KUKA KRL program: MyProgram_317().src

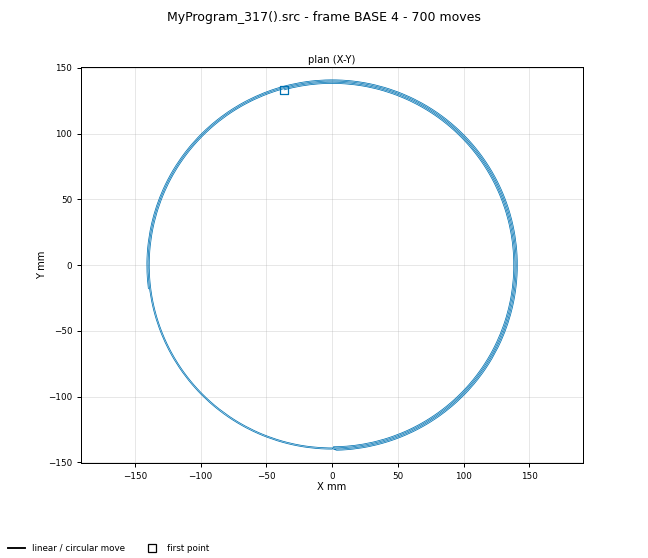
[picture p0: tool path of MyProgram_317().src in frame BASE 4, 700 of 700 moves have a stored position in this frame; points joined in program order, loops and branches not executed]
&ACCESS RVP
&REL 1
&PARAM TEMPLATE = C:\KRC\Roboter\Template\vorgabe
&PARAM EDITMASK = *
DEF MyProgram_317()
; ---- Setting reference (Base) ----
$BASE = BASE_DATA[4]

; --------------------------
; ---- Setting tool (TCP) ----
$TOOL = TOOL_DATA[3]
; --------------------------

$VEL.CP = VEL_APROX_PRINT
Startdeposition()
$VEL.CP = VEL_PRINT
LIN {X -36.4177,Y 133.3267,Z 184,A 105.8748,B 3.6775,C 0.0605,E1 3.6399,E2 347.4823} C_DIS
LIN {X -33.6227,Y 134.0568,Z 184,A 104.6666,B 3.6776,C 0.0598,E1 3.6432,E2 348.691} C_DIS
LIN {X -29.9714,Y 134.9221,Z 184,A 103.1035,B 3.6776,C 0.059,E1 3.6474,E2 350.2543} C_DIS
LIN {X -26.7547,Y 135.5966,Z 184,A 101.734,B 3.6776,C 0.0584,E1 3.6512,E2 351.6239} C_DIS
LIN {X -23.5921,Y 136.1822,Z 184,A 100.3951,B 3.6776,C 0.0579,E1 3.6549,E2 352.9627} C_DIS
LIN {X -20.3485,Y 136.7048,Z 184,A 99.029,B 3.6776,C 0.0575,E1 3.6586,E2 354.3286} C_DIS
LIN {X -17.2099,Y 137.135,Z 184,A 97.7126,B 3.6776,C 0.0572,E1 3.6623,E2 355.6447} C_DIS
LIN {X -14.2664,Y 137.4713,Z 184,A 96.4709,B 3.6776,C 0.057,E1 3.6657,E2 356.8874} C_DIS
LIN {X -10.8915,Y 137.7809,Z 184,A 95.0782,B 3.6776,C 0.0567,E1 3.6696,E2 358.278} C_DIS
LIN {X -7.7622,Y 137.9925,Z 184,A 93.7791,B 3.6776,C 0.0566,E1 3.6732,E2 359.5763} C_DIS
LIN {X -3.6918,Y 138.1595,Z 184,A 92.0273,B 3.6776,C 0.0571,E1 3.6781,E2 361.3349} C_DIS
LIN {X 0,Y 138.2109,Z 184,A 90.5659,B 3.6776,C 0.0566,E1 3.6822,E2 362.7873} C_DIS
LIN {X 3.0237,Y 138.1776,Z 184,A 89.3114,B 3.6776,C 0.0568,E1 3.6857,E2 364.0415} C_DIS
LIN {X 6.1171,Y 138.0752,Z 184,A 88.0293,B 3.6776,C 0.0571,E1 3.6893,E2 365.3229} C_DIS
LIN {X 10.3123,Y 137.8236,Z 184,A 86.2404,B 3.6776,C 0.0579,E1 3.6943,E2 367.1167} C_DIS
LIN {X 13.9962,Y 137.5004,Z 184,A 84.7627,B 3.6776,C 0.058,E1 3.6984,E2 368.5872} C_DIS
LIN {X 17.1189,Y 137.1464,Z 184,A 83.4643,B 3.6776,C 0.0585,E1 3.702,E2 369.8846} C_DIS
LIN {X 20.3485,Y 136.7048,Z 184,A 82.1206,B 3.6776,C 0.0591,E1 3.7057,E2 371.227} C_DIS
LIN {X 23.0597,Y 136.2716,Z 184,A 80.9465,B 3.6776,C 0.0601,E1 3.7089,E2 372.405} C_DIS
LIN {X 26.7088,Y 135.6054,Z 184,A 79.462,B 3.6776,C 0.0606,E1 3.713,E2 373.8826} C_DIS
LIN {X 29.9253,Y 134.932,Z 184,A 78.1102,B 3.6776,C 0.0614,E1 3.7167,E2 375.2327} C_DIS
LIN {X 32.8099,Y 134.2582,Z 184,A 76.899,B 3.6776,C 0.0622,E1 3.72,E2 376.4414} C_DIS
LIN {X 35.9709,Y 133.4458,Z 184,A 75.5188,B 3.6776,C 0.0635,E1 3.7237,E2 377.8247} C_DIS
LIN {X 39.6415,Y 132.404,Z 184,A 73.9879,B 3.6776,C 0.0644,E1 3.7278,E2 379.3491} C_DIS
LIN {X 42.8155,Y 131.4116,Z 184,A 72.6248,B 3.6776,C 0.0656,E1 3.7314,E2 380.7099} C_DIS
LIN {X 45.6313,Y 130.4587,Z 184,A 71.4074,B 3.6775,C 0.0667,E1 3.7346,E2 381.9252} C_DIS
LIN {X 49.2779,Y 129.1276,Z 184,A 69.8203,B 3.6775,C 0.0682,E1 3.7388,E2 383.5094} C_DIS
LIN {X 52.4222,Y 127.8831,Z 184,A 68.4385,B 3.6775,C 0.0696,E1 3.7424,E2 384.8886} C_DIS
LIN {X 55.1838,Y 126.7138,Z 184,A 67.1766,B 3.6774,C 0.0713,E1 3.7456,E2 386.1525} C_DIS
LIN {X 58.7493,Y 125.1027,Z 184,A 65.6176,B 3.6774,C 0.0727,E1 3.7495,E2 387.7036} C_DIS
LIN {X 61.8796,Y 123.5843,Z 184,A 64.203,B 3.6774,C 0.0744,E1 3.7531,E2 389.1147} C_DIS
LIN {X 64.8421,Y 122.0551,Z 184,A 62.835,B 3.6773,C 0.0761,E1 3.7565,E2 390.4809} C_DIS
LIN {X 68.469,Y 120.0586,Z 184,A 61.0927,B 3.6773,C 0.0789,E1 3.7607,E2 392.2263} C_DIS
LIN {X 71.8734,Y 118.0527,Z 184,A 59.5538,B 3.6773,C 0.0804,E1 3.7644,E2 393.753} C_DIS
LIN {X 74.8883,Y 116.1637,Z 184,A 58.1092,B 3.6772,C 0.0824,E1 3.7678,E2 395.1939} C_DIS
LIN {X 77.8197,Y 114.2206,Z 184,A 56.6827,B 3.6772,C 0.0845,E1 3.7711,E2 396.6165} C_DIS
LIN {X 80.7488,Y 112.169,Z 184,A 55.2381,B 3.6771,C 0.0867,E1 3.7744,E2 398.0564} C_DIS
LIN {X 83.9195,Y 109.8161,Z 184,A 53.5602,B 3.677,C 0.0899,E1 3.7781,E2 399.7395} C_DIS
LIN {X 87.1141,Y 107.3005,Z 184,A 51.9899,B 3.677,C 0.0918,E1 3.7815,E2 401.2957} C_DIS
LIN {X 90.0725,Y 104.8286,Z 184,A 50.3385,B 3.6769,C 0.0954,E1 3.7851,E2 402.9538} C_DIS
LIN {X 93.2043,Y 102.055,Z 184,A 48.7445,B 3.6769,C 0.0973,E1 3.7883,E2 404.5307} C_DIS
LIN {X 95.7956,Y 99.6265,Z 184,A 47.3082,B 3.6767,C 0.0999,E1 3.7912,E2 405.9628} C_DIS
LIN {X 98.6354,Y 96.8148,Z 184,A 45.6237,B 3.6767,C 0.1035,E1 3.7946,E2 407.6509} C_DIS
LIN {X 101.4499,Y 93.8625,Z 184,A 44.0571,B 3.6766,C 0.1058,E1 3.7975,E2 409.2025} C_DIS
LIN {X 104.0652,Y 90.9534,Z 184,A 42.3981,B 3.6765,C 0.1097,E1 3.8006,E2 410.8664} C_DIS
LIN {X 106.7196,Y 87.8247,Z 184,A 40.8296,B 3.6764,C 0.112,E1 3.8034,E2 412.4188} C_DIS
LIN {X 108.9505,Y 85.0413,Z 184,A 39.4004,B 3.6763,C 0.1148,E1 3.8059,E2 413.8423} C_DIS
LIN {X 111.2875,Y 81.9584,Z 184,A 37.7496,B 3.6762,C 0.119,E1 3.8086,E2 415.4993} C_DIS
LIN {X 113.7044,Y 78.572,Z 184,A 36.1718,B 3.6761,C 0.1215,E1 3.8111,E2 417.0593} C_DIS
LIN {X 115.668,Y 75.6515,Z 184,A 34.6865,B 3.676,C 0.1252,E1 3.8134,E2 418.5484} C_DIS
LIN {X 118.0397,Y 71.895,Z 184,A 32.9814,B 3.6759,C 0.1282,E1 3.8159,E2 420.237} C_DIS
LIN {X 119.8206,Y 68.8859,Z 184,A 31.5781,B 3.6757,C 0.1313,E1 3.8179,E2 421.635} C_DIS
LIN {X 121.5433,Y 65.7989,Z 184,A 30.0427,B 3.6756,C 0.1357,E1 3.82,E2 423.1798} C_DIS
LIN {X 123.5623,Y 61.9243,Z 184,A 28.4136,B 3.6755,C 0.1383,E1 3.822,E2 424.7867} C_DIS
LIN {X 125.0605,Y 58.8392,Z 184,A 27.0414,B 3.6754,C 0.1414,E1 3.8237,E2 426.1533} C_DIS
LIN {X 126.3707,Y 55.9663,Z 184,A 25.7977,B 3.6753,C 0.1441,E1 3.8251,E2 427.3892} C_DIS
LIN {X 127.7,Y 52.8622,Z 184,A 24.3996,B 3.6751,C 0.1477,E1 3.8266,E2 428.7878} C_DIS
LIN {X 129.1276,Y 49.2779,Z 184,A 22.8878,B 3.675,C 0.151,E1 3.8281,E2 430.2893} C_DIS
LIN {X 130.2884,Y 46.1206,Z 184,A 21.5479,B 3.6749,C 0.1541,E1 3.8294,E2 431.6229} C_DIS
LIN {X 131.2362,Y 43.3441,Z 184,A 20.3532,B 3.6747,C 0.1571,E1 3.8304,E2 432.8155} C_DIS
LIN {X 132.404,Y 39.6415,Z 184,A 18.8234,B 3.6746,C 0.1606,E1 3.8317,E2 434.3361} C_DIS
LIN {X 133.3267,Y 36.4177,Z 184,A 17.4858,B 3.6744,C 0.1638,E1 3.8327,E2 435.6678} C_DIS
LIN {X 134.0348,Y 33.7096,Z 184,A 16.324,B 3.6743,C 0.167,E1 3.8335,E2 436.8304} C_DIS
LIN {X 134.9221,Y 29.9714,Z 184,A 14.837,B 3.6742,C 0.1702,E1 3.8344,E2 438.3049} C_DIS
LIN {X 135.5966,Y 26.7547,Z 184,A 13.5266,B 3.674,C 0.1734,E1 3.8352,E2 439.6095} C_DIS
LIN {X 136.1822,Y 23.5921,Z 184,A 12.2445,B 3.6739,C 0.1765,E1 3.8358,E2 440.8858} C_DIS
LIN {X 136.7048,Y 20.3485,Z 184,A 10.9352,B 3.6737,C 0.1797,E1 3.8363,E2 442.1892} C_DIS
LIN {X 137.0724,Y 17.6872,Z 184,A 9.8194,B 3.6735,C 0.1829,E1 3.8368,E2 443.3059} C_DIS
LIN {X 137.4956,Y 14.0415,Z 184,A 8.4072,B 3.6734,C 0.1859,E1 3.8372,E2 444.7052} C_DIS
LIN {X 137.7809,Y 10.8915,Z 184,A 7.1428,B 3.6732,C 0.1891,E1 3.8375,E2 445.9645} C_DIS
LIN {X 137.9925,Y 7.7622,Z 184,A 5.9051,B 3.6731,C 0.192,E1 3.8377,E2 447.195} C_DIS
LIN {X 138.1604,Y 3.6595,Z 184,A 4.2009,B 3.6728,C 0.1969,E1 3.8379,E2 448.9004} C_DIS
LIN {X 138.2105,Y 0,Z 184,A 2.8172,B 3.6727,C 0.1996,E1 3.8379,E2 450.2682} C_DIS
LIN {X 138.1769,Y -3.0677,Z 184,A 1.5727,B 3.6725,C 0.2029,E1 3.8379,E2 451.51} C_DIS
LIN {X 138.0752,Y -6.1171,Z 184,A 0.3524,B 3.6723,C 0.206,E1 3.8377,E2 452.7255} C_DIS
LIN {X 137.8237,Y -10.3111,Z 184,A -1.3754,B 3.6721,C 0.2107,E1 3.8374,E2 454.4526} C_DIS
LIN {X 137.5004,Y -13.9962,Z 184,A -2.8057,B 3.6719,C 0.2139,E1 3.837,E2 455.8708} C_DIS
LIN {X 137.1464,Y -17.1189,Z 184,A -4.063,B 3.6717,C 0.217,E1 3.8366,E2 457.1232} C_DIS
LIN {X 136.7048,Y -20.3485,Z 184,A -5.3655,B 3.6715,C 0.2203,E1 3.8361,E2 458.4205} C_DIS
LIN {X 136.2752,Y -23.0383,Z 184,A -6.4989,B 3.6713,C 0.2235,E1 3.8356,E2 459.5551} C_DIS
LIN {X 135.6054,Y -26.7088,Z 184,A -7.9465,B 3.6711,C 0.2267,E1 3.8348,E2 460.9911} C_DIS
LIN {X 134.932,Y -29.9253,Z 184,A -9.2568,B 3.6709,C 0.2299,E1 3.8341,E2 462.2958} C_DIS
LIN {X 134.1769,Y -33.1472,Z 184,A -10.5844,B 3.6707,C 0.2332,E1 3.8332,E2 463.6187} C_DIS
LIN {X 133.4627,Y -35.9077,Z 184,A -11.7334,B 3.6705,C 0.236,E1 3.8324,E2 464.7642} C_DIS
LIN {X 132.4869,Y -39.3583,Z 184,A -13.1732,B 3.6703,C 0.2396,E1 3.8313,E2 466.1992} C_DIS
LIN {X 131.4116,Y -42.8155,Z 184,A -14.6088,B 3.6701,C 0.2429,E1 3.8301,E2 467.6275} C_DIS
LIN {X 130.3049,Y -46.0747,Z 184,A -15.9862,B 3.6699,C 0.2462,E1 3.8288,E2 468.9996} C_DIS
LIN {X 129.1276,Y -49.2779,Z 184,A -17.3523,B 3.6696,C 0.2494,E1 3.8275,E2 470.3606} C_DIS
LIN {X 127.9871,Y -52.1642,Z 184,A -18.6113,B 3.6694,C 0.2525,E1 3.8262,E2 471.617} C_DIS
LIN {X 126.5358,Y -55.5957,Z 184,A -20.0872,B 3.6692,C 0.2558,E1 3.8246,E2 473.0852} C_DIS
LIN {X 125.276,Y -58.3747,Z 184,A -21.3124,B 3.669,C 0.2586,E1 3.8231,E2 474.3062} C_DIS
LIN {X 123.5843,Y -61.8796,Z 184,A -22.8693,B 3.6687,C 0.2621,E1 3.8212,E2 475.8571} C_DIS
LIN {X 121.9809,Y -64.9833,Z 184,A -24.2702,B 3.6685,C 0.2653,E1 3.8194,E2 477.2531} C_DIS
LIN {X 120.2686,Y -68.1009,Z 184,A -25.6961,B 3.6683,C 0.2685,E1 3.8175,E2 478.6738} C_DIS
LIN {X 118.5194,Y -71.1011,Z 184,A -27.1792,B 3.668,C 0.2725,E1 3.8154,E2 480.1638} C_DIS
LIN {X 116.1637,Y -74.8883,Z 184,A -28.8795,B 3.6678,C 0.2754,E1 3.8128,E2 481.8462} C_DIS
LIN {X 114.2206,Y -77.8197,Z 184,A -30.2911,B 3.6676,C 0.2784,E1 3.8107,E2 483.253} C_DIS
LIN {X 112.169,Y -80.7488,Z 184,A -31.7282,B 3.6673,C 0.2814,E1 3.8083,E2 484.6853} C_DIS
LIN {X 109.8667,Y -83.8533,Z 184,A -33.3715,B 3.667,C 0.2855,E1 3.8056,E2 486.3352} C_DIS
LIN {X 107.3005,Y -87.1141,Z 184,A -35.0216,B 3.6668,C 0.2887,E1 3.8027,E2 487.9776} C_DIS
LIN {X 104.4481,Y -90.5143,Z 184,A -36.7357,B 3.6665,C 0.2914,E1 3.7996,E2 489.6767} C_DIS
LIN {X 102.055,Y -93.2043,Z 184,A -38.2644,B 3.6663,C 0.295,E1 3.7968,E2 491.2114} C_DIS
LIN {X 98.9867,Y -96.4567,Z 184,A -40.0606,B 3.666,C 0.2983,E1 3.7933,E2 493.0015} C_DIS
LIN {X 95.8325,Y -99.591,Z 184,A -41.7813,B 3.6658,C 0.3008,E1 3.7899,E2 494.7077} C_DIS
LIN {X 93.2043,Y -102.055,Z 184,A -43.2299,B 3.6656,C 0.3033,E1 3.7869,E2 496.1515} C_DIS
LIN {X 90.1903,Y -104.7271,Z 184,A -44.9204,B 3.6653,C 0.3068,E1 3.7834,E2 497.846} C_DIS
LIN {X 87.1339,Y -107.2843,Z 184,A -46.4677,B 3.6651,C 0.3088,E1 3.7801,E2 499.3809} C_DIS
LIN {X 84.317,Y -109.5121,Z 184,A -47.9844,B 3.6649,C 0.3118,E1 3.7767,E2 500.9024} C_DIS
LIN {X 80.7694,Y -112.1541,Z 184,A -49.6964,B 3.6647,C 0.3138,E1 3.7729,E2 502.5998} C_DIS
LIN {X 77.8407,Y -114.2063,Z 184,A -51.1541,B 3.6645,C 0.3161,E1 3.7695,E2 504.0554} C_DIS
LIN {X 74.8883,Y -116.1637,Z 184,A -52.5889,B 3.6643,C 0.3182,E1 3.7662,E2 505.4868} C_DIS
LIN {X 71.895,Y -118.0397,Z 184,A -54.0208,B 3.6641,C 0.3202,E1 3.7628,E2 506.9156} C_DIS
LIN {X 68.8859,Y -119.8206,Z 184,A -55.4417,B 3.664,C 0.3221,E1 3.7594,E2 508.3337} C_DIS
LIN {X 65.6732,Y -121.6108,Z 184,A -57.0582,B 3.6637,C 0.3253,E1 3.7554,E2 509.9635} C_DIS
LIN {X 61.9243,Y -123.5623,Z 184,A -58.6521,B 3.6637,C 0.3262,E1 3.7515,E2 511.5378} C_DIS
LIN {X 58.8392,Y -125.0605,Z 184,A -60.0471,B 3.6635,C 0.3278,E1 3.748,E2 512.9302} C_DIS
LIN {X 55.641,Y -126.5161,Z 184,A -61.4766,B 3.6633,C 0.3294,E1 3.7443,E2 514.3572} C_DIS
LIN {X 52.4678,Y -127.8647,Z 184,A -62.881,B 3.6632,C 0.3309,E1 3.7407,E2 515.7593} C_DIS
LIN {X 49.2779,Y -129.1276,Z 184,A -64.2795,B 3.6631,C 0.3323,E1 3.7371,E2 517.1556} C_DIS
LIN {X 46.1206,Y -130.2884,Z 184,A -65.6513,B 3.6629,C 0.3336,E1 3.7335,E2 518.5253} C_DIS
LIN {X 43.3085,Y -131.2481,Z 184,A -66.8658,B 3.6629,C 0.3347,E1 3.7303,E2 519.7384} C_DIS
LIN {X 39.6415,Y -132.404,Z 184,A -68.4354,B 3.6627,C 0.336,E1 3.7261,E2 521.3058} C_DIS
LIN {X 36.4177,Y -133.3267,Z 184,A -69.8062,B 3.6627,C 0.3371,E1 3.7224,E2 522.675} C_DIS
LIN {X 33.1934,Y -134.1658,Z 184,A -71.1697,B 3.6625,C 0.3381,E1 3.7187,E2 524.037} C_DIS
LIN {X 30.4533,Y -134.812,Z 184,A -72.3636,B 3.6625,C 0.3392,E1 3.7154,E2 525.2351} C_DIS
LIN {X 26.7547,Y -135.5966,Z 184,A -73.8726,B 3.6624,C 0.3398,E1 3.7113,E2 526.7373} C_DIS
LIN {X 23.5921,Y -136.1822,Z 184,A -75.1907,B 3.6624,C 0.3405,E1 3.7077,E2 528.0542} C_DIS
LIN {X 20.3485,Y -136.7048,Z 184,A -76.541,B 3.6622,C 0.3412,E1 3.704,E2 529.4037} C_DIS
LIN {X 17.2099,Y -137.135,Z 184,A -77.8367,B 3.6622,C 0.3417,E1 3.7004,E2 530.6977} C_DIS
LIN {X 14.5476,Y -137.4411,Z 184,A -78.9933,B 3.6622,C 0.3426,E1 3.6971,E2 531.861} C_DIS
LIN {X 10.8915,Y -137.7809,Z 184,A -80.4558,B 3.6622,C 0.3427,E1 3.6931,E2 533.3165} C_DIS
LIN {X 7.7622,Y -137.9925,Z 184,A -81.7476,B 3.6621,C 0.3431,E1 3.6895,E2 534.6078} C_DIS
LIN {X 4.6115,Y -138.134,Z 184,A -83.048,B 3.6621,C 0.3433,E1 3.6859,E2 535.9079} C_DIS
LIN {X 0.9865,Y -138.204,Z 184,A -84.071,B 3.6624,C 0.3395,E1 3.6832,E2 536.8675} C_DIS
Enddeposition()
LIN {X 0.9865,Y -138.204,Z 184,A -84.071,B 3.6624,C 0.3395,E1 3.6832,E2 536.8675} C_DIS
Startdeposition()
$VEL.CP = VEL_PRINT
LIN {X 1.6267,Y -139.1018,Z 184,A -83.626,B 3.6446,C 0.3393,E1 3.6667,E2 536.434} C_DIS
LIN {X 4.5561,Y -139.0367,Z 184,A -82.3295,B 3.6447,C 0.3382,E1 3.6703,E2 535.1247} C_DIS
LIN {X 8.311,Y -138.8613,Z 184,A -81.0351,B 3.6446,C 0.34,E1 3.6738,E2 533.8639} C_DIS
LIN {X 11.0661,Y -138.6702,Z 184,A -79.683,B 3.6448,C 0.3376,E1 3.6777,E2 532.4822} C_DIS
LIN {X 14.8601,Y -138.3135,Z 184,A -78.2274,B 3.6448,C 0.338,E1 3.6817,E2 531.0411} C_DIS
LIN {X 22.3175,Y -137.3087,Z 184,A -75.1897,B 3.6448,C 0.3369,E1 3.6901,E2 528.0102} C_DIS
LIN {X 27.2301,Y -136.4192,Z 184,A -73.0374,B 3.6451,C 0.3346,E1 3.696,E2 525.8436} C_DIS
LIN {X 31.257,Y -135.5525,Z 184,A -71.0765,B 3.6454,C 0.3308,E1 3.7015,E2 523.8458} C_DIS
LIN {X 34.8949,Y -134.6633,Z 184,A -69.7728,B 3.6454,C 0.3318,E1 3.7049,E2 522.5736} C_DIS
LIN {X 38.7466,Y -133.6046,Z 184,A -68.4032,B 3.6452,C 0.3329,E1 3.7085,E2 521.2402} C_DIS
LIN {X 42.0447,Y -132.6035,Z 184,A -66.8695,B 3.6454,C 0.3305,E1 3.7127,E2 519.6902} C_DIS
LIN {X 45.813,Y -131.3491,Z 184,A -64.552,B 3.6462,C 0.3221,E1 3.719,E2 517.2789} C_DIS
LIN {X 51.2002,Y -129.346,Z 184,A -62.7921,B 3.6459,C 0.3253,E1 3.7234,E2 515.6001} C_DIS
LIN {X 54.8124,Y -127.8558,Z 184,A -61.4097,B 3.6459,C 0.3256,E1 3.7269,E2 514.2473} C_DIS
LIN {X 57.5864,Y -126.6329,Z 184,A -59.9335,B 3.6462,C 0.3218,E1 3.7307,E2 512.7395} C_DIS
LIN {X 60.8952,Y -125.0744,Z 184,A -58.6873,B 3.6462,C 0.3223,E1 3.7338,E2 511.5274} C_DIS
LIN {X 63.9287,Y -123.5522,Z 184,A -57.1271,B 3.6465,C 0.3187,E1 3.7377,E2 509.9442} C_DIS
LIN {X 67.7295,Y -121.5103,Z 184,A -55.4455,B 3.6466,C 0.3171,E1 3.7418,E2 508.2743} C_DIS
LIN {X 71.3493,Y -119.4202,Z 184,A -53.9193,B 3.6466,C 0.3164,E1 3.7454,E2 506.7731} C_DIS
LIN {X 75.2493,Y -117.0022,Z 184,A -51.9472,B 3.647,C 0.3126,E1 3.7501,E2 504.7885} C_DIS
LIN {X 78.5811,Y -114.7908,Z 184,A -50.3195,B 3.6472,C 0.31,E1 3.7539,E2 503.1621} C_DIS
LIN {X 81.9197,Y -112.433,Z 184,A -48.5917,B 3.6475,C 0.3066,E1 3.7578,E2 501.427} C_DIS
LIN {X 86.4283,Y -109.0051,Z 184,A -46.356,B 3.6478,C 0.3033,E1 3.7627,E2 499.2025} C_DIS
LIN {X 89.6043,Y -106.4097,Z 184,A -44.7166,B 3.648,C 0.3007,E1 3.7662,E2 497.5686} C_DIS
LIN {X 92.8185,Y -103.6176,Z 184,A -43.0112,B 3.6483,C 0.2977,E1 3.7698,E2 495.8682} C_DIS
LIN {X 96.4701,Y -100.2276,Z 184,A -41.08,B 3.6485,C 0.2949,E1 3.7737,E2 493.9516} C_DIS
LIN {X 99.1485,Y -97.5783,Z 184,A -39.5527,B 3.6487,C 0.2919,E1 3.7767,E2 492.4263} C_DIS
LIN {X 101.875,Y -94.7279,Z 184,A -37.9879,B 3.6489,C 0.2891,E1 3.7797,E2 490.8682} C_DIS
LIN {X 104.0406,Y -92.3445,Z 184,A -36.5334,B 3.6493,C 0.2848,E1 3.7824,E2 489.3954} C_DIS
LIN {X 107.3985,Y -88.4172,Z 184,A -34.5568,B 3.6495,C 0.2818,E1 3.7859,E2 487.4374} C_DIS
LIN {X 110.2779,Y -84.7985,Z 184,A -32.9995,B 3.6495,C 0.2812,E1 3.7886,E2 485.925} C_DIS
LIN {X 113.183,Y -80.8795,Z 184,A -30.7961,B 3.6501,C 0.2744,E1 3.7922,E2 483.694} C_DIS
LIN {X 115.3285,Y -77.79,Z 184,A -29.2513,B 3.6504,C 0.2707,E1 3.7947,E2 482.1486} C_DIS
LIN {X 117.9246,Y -73.7956,Z 184,A -27.3604,B 3.6506,C 0.2668,E1 3.7975,E2 480.2656} C_DIS
LIN {X 120.0287,Y -70.3209,Z 184,A -25.5164,B 3.6511,C 0.2607,E1 3.8001,E2 478.3973} C_DIS
LIN {X 121.8673,Y -67.0847,Z 184,A -24.3462,B 3.6511,C 0.2609,E1 3.8017,E2 477.2744} C_DIS
LIN {X 123.5248,Y -63.9809,Z 184,A -22.7776,B 3.6514,C 0.2559,E1 3.8037,E2 475.6887} C_DIS
LIN {X 125.4873,Y -60.0356,Z 184,A -21.2126,B 3.6516,C 0.2541,E1 3.8056,E2 474.1553} C_DIS
LIN {X 127.2516,Y -56.2031,Z 184,A -19.4239,B 3.6519,C 0.249,E1 3.8076,E2 472.3585} C_DIS
LIN {X 128.9238,Y -52.25,Z 184,A -17.8419,B 3.6521,C 0.2464,E1 3.8093,E2 470.7998} C_DIS
LIN {X 129.9917,Y -49.5393,Z 184,A -16.3578,B 3.6525,C 0.24,E1 3.8108,E2 469.277} C_DIS
LIN {X 131.2146,Y -46.2011,Z 184,A -15.1434,B 3.6525,C 0.2389,E1 3.8119,E2 468.0946} C_DIS
LIN {X 132.3294,Y -42.9028,Z 184,A -13.9835,B 3.6526,C 0.2381,E1 3.8129,E2 466.9699} C_DIS
LIN {X 133.423,Y -39.3669,Z 184,A -12.4,B 3.6529,C 0.2333,E1 3.8142,E2 465.3774} C_DIS
LIN {X 134.2134,Y -36.5889,Z 184,A -11.3088,B 3.6531,C 0.2312,E1 3.815,E2 464.2983} C_DIS
LIN {X 135.1389,Y -33.0005,Z 184,A -9.7166,B 3.6534,C 0.2262,E1 3.8161,E2 462.6962} C_DIS
LIN {X 136.8507,Y -24.9703,Z 184,A -6.558,B 3.6538,C 0.2194,E1 3.8179,E2 459.5646} C_DIS
LIN {X 137.8292,Y -18.845,Z 184,A -3.9527,B 3.6543,C 0.2117,E1 3.819,E2 456.9508} C_DIS
LIN {X 138.2931,Y -15.0497,Z 184,A -2.6362,B 3.6543,C 0.2102,E1 3.8194,E2 455.667} C_DIS
LIN {X 138.6077,Y -11.8054,Z 184,A -1.2782,B 3.6546,C 0.2062,E1 3.8197,E2 454.3061} C_DIS
LIN {X 138.8743,Y -8.0994,Z 184,A 0.3268,B 3.6549,C 0.2011,E1 3.82,E2 452.6903} C_DIS
LIN {X 139.0413,Y -4.39,Z 184,A 1.5468,B 3.6549,C 0.2003,E1 3.8201,E2 451.5097} C_DIS
LIN {X 139.1063,Y -0.9898,Z 184,A 3.0194,B 3.6552,C 0.1955,E1 3.8201,E2 450.0267} C_DIS
LIN {X 139.0868,Y 2.5321,Z 184,A 4.4683,B 3.6554,C 0.1914,E1 3.8201,E2 448.577} C_DIS
LIN {X 138.9387,Y 6.8925,Z 184,A 6.1187,B 3.6555,C 0.188,E1 3.8199,E2 446.9445} C_DIS
LIN {X 138.7685,Y 9.7424,Z 184,A 7.2364,B 3.6557,C 0.1854,E1 3.8197,E2 445.8337} C_DIS
LIN {X 138.4021,Y 14.031,Z 184,A 9.0908,B 3.656,C 0.1795,E1 3.8193,E2 443.9676} C_DIS
LIN {X 137.8074,Y 19.0003,Z 184,A 11.021,B 3.6562,C 0.1752,E1 3.8186,E2 442.0532} C_DIS
LIN {X 136.6868,Y 25.8495,Z 184,A 13.7424,B 3.6565,C 0.1688,E1 3.8173,E2 439.3479} C_DIS
LIN {X 135.7284,Y 30.4871,Z 184,A 15.6833,B 3.6567,C 0.1635,E1 3.8162,E2 437.4072} C_DIS
LIN {X 134.8596,Y 34.1218,Z 184,A 17.0595,B 3.6568,C 0.1611,E1 3.8153,E2 436.0513} C_DIS
LIN {X 133.9801,Y 37.4261,Z 184,A 18.3557,B 3.6569,C 0.1585,E1 3.8143,E2 434.7687} C_DIS
LIN {X 133.1804,Y 40.1828,Z 184,A 19.6449,B 3.6571,C 0.1541,E1 3.8133,E2 433.4652} C_DIS
LIN {X 132.0698,Y 43.6921,Z 184,A 21.0366,B 3.6572,C 0.1514,E1 3.8121,E2 432.0887} C_DIS
LIN {X 131.1049,Y 46.5121,Z 184,A 22.1652,B 3.6573,C 0.1493,E1 3.8111,E2 430.9723} C_DIS
LIN {X 129.8289,Y 49.9603,Z 184,A 23.702,B 3.6575,C 0.145,E1 3.8095,E2 429.4319} C_DIS
LIN {X 128.518,Y 53.2411,Z 184,A 25.1194,B 3.6576,C 0.1416,E1 3.8081,E2 428.0187} C_DIS
LIN {X 127.0919,Y 56.5602,Z 184,A 26.5206,B 3.6577,C 0.1387,E1 3.8065,E2 426.6279} C_DIS
LIN {X 125.8669,Y 59.241,Z 184,A 27.6711,B 3.6578,C 0.1363,E1 3.8052,E2 425.4851} C_DIS
LIN {X 124.2392,Y 62.5804,Z 184,A 29.2061,B 3.658,C 0.1323,E1 3.8032,E2 423.9489} C_DIS
LIN {X 122.3439,Y 66.2122,Z 184,A 30.8919,B 3.6581,C 0.1281,E1 3.801,E2 422.2627} C_DIS
LIN {X 120.2591,Y 69.9265,Z 184,A 32.5879,B 3.6583,C 0.1244,E1 3.7987,E2 420.5735} C_DIS
LIN {X 117.9197,Y 73.8036,Z 184,A 34.407,B 3.6583,C 0.1204,E1 3.796,E2 418.7597} C_DIS
LIN {X 115.4373,Y 77.6292,Z 184,A 36.2311,B 3.6585,C 0.1165,E1 3.7932,E2 416.9419} C_DIS
LIN {X 112.8595,Y 81.3312,Z 184,A 38.0454,B 3.6586,C 0.1126,E1 3.7903,E2 415.1326} C_DIS
LIN {X 110.3375,Y 84.7206,Z 184,A 40.762,B 3.6591,C 0.0983,E1 3.7855,E2 412.29} C_DIS
LIN {X 105.0956,Y 91.1426,Z 184,A 43.1443,B 3.659,C 0.1018,E1 3.7814,E2 410.0398} C_DIS
LIN {X 101.7038,Y 94.9118,Z 184,A 45.037,B 3.659,C 0.0994,E1 3.7778,E2 408.1715} C_DIS
LIN {X 98.4714,Y 98.2617,Z 184,A 46.909,B 3.6591,C 0.0959,E1 3.7742,E2 406.305} C_DIS
LIN {X 96.221,Y 100.4661,Z 184,A 48.7641,B 3.6593,C 0.0876,E1 3.7703,E2 404.3788} C_DIS
LIN {X 92.093,Y 104.2629,Z 184,A 50.4182,B 3.6593,C 0.0899,E1 3.767,E2 402.8079} C_DIS
LIN {X 88.23,Y 107.5519,Z 184,A 52.4688,B 3.6593,C 0.0864,E1 3.7626,E2 400.762} C_DIS
LIN {X 84.5498,Y 110.4682,Z 184,A 54.3314,B 3.6594,C 0.0836,E1 3.7585,E2 398.9083} C_DIS
LIN {X 81.5522,Y 112.6993,Z 184,A 56.4543,B 3.6596,C 0.0751,E1 3.7536,E2 396.7114} C_DIS
LIN {X 76.8945,Y 115.9272,Z 184,A 58.1486,B 3.6596,C 0.0777,E1 3.7498,E2 395.0982} C_DIS
LIN {X 73.4331,Y 118.1502,Z 184,A 59.7449,B 3.6596,C 0.076,E1 3.7461,E2 393.5143} C_DIS
LIN {X 69.8491,Y 120.3039,Z 184,A 61.4765,B 3.6596,C 0.0733,E1 3.7419,E2 391.7815} C_DIS
LIN {X 65.8036,Y 122.5634,Z 184,A 63.3616,B 3.6596,C 0.0708,E1 3.7373,E2 389.8994} C_DIS
LIN {X 63.0762,Y 123.9868,Z 184,A 65.1665,B 3.6598,C 0.064,E1 3.7326,E2 388.0267} C_DIS
LIN {X 58.1292,Y 126.382,Z 184,A 66.826,B 3.6598,C 0.0668,E1 3.7286,E2 386.4438} C_DIS
LIN {X 53.9781,Y 128.2102,Z 184,A 68.4391,B 3.6598,C 0.067,E1 3.7246,E2 384.8628} C_DIS
LIN {X 51.4322,Y 129.2534,Z 184,A 69.7852,B 3.6598,C 0.0637,E1 3.721,E2 383.4903} C_DIS
LIN {X 47.4222,Y 130.7767,Z 184,A 71.4346,B 3.6598,C 0.0629,E1 3.7167,E2 381.8559} C_DIS
LIN {X 42.7659,Y 132.3731,Z 184,A 73.2656,B 3.6598,C 0.0627,E1 3.7119,E2 380.0499} C_DIS
LIN {X 39.1536,Y 133.4855,Z 184,A 74.85,B 3.6598,C 0.061,E1 3.7077,E2 378.4624} C_DIS
LIN {X 36.3496,Y 134.2772,Z 184,A 76.1941,B 3.6598,C 0.0587,E1 3.704,E2 377.1006} C_DIS
LIN {X 33.0187,Y 135.1345,Z 184,A 77.5771,B 3.6599,C 0.0579,E1 3.7003,E2 375.7222} C_DIS
LIN {X 24.4171,Y 136.9497,Z 184,A 81.1038,B 3.6599,C 0.0564,E1 3.6907,E2 372.2085} C_DIS
LIN {X 18.0552,Y 137.9328,Z 184,A 83.6491,B 3.6599,C 0.056,E1 3.6837,E2 369.6773} C_DIS
LIN {X 15.6018,Y 138.2337,Z 184,A 84.8854,B 3.6599,C 0.0537,E1 3.6802,E2 368.4143} C_DIS
LIN {X 11.7127,Y 138.6155,Z 184,A 86.3851,B 3.6599,C 0.0541,E1 3.676,E2 366.9288} C_DIS
LIN {X 7.8041,Y 138.8925,Z 184,A 87.9522,B 3.6599,C 0.0541,E1 3.6717,E2 365.3682} C_DIS
LIN {X 3.8245,Y 139.057,Z 184,A 89.6538,B 3.6599,C 0.0532,E1 3.6669,E2 363.6596} C_DIS
LIN {X 0.0191,Y 139.1116,Z 184,A 91.3045,B 3.6599,C 0.0523,E1 3.6623,E2 361.9993} C_DIS
LIN {X -3.784,Y 139.0582,Z 184,A 92.7529,B 3.6599,C 0.0532,E1 3.6583,E2 360.5662} C_DIS
LIN {X -10.3027,Y 138.7276,Z 184,A 95.4954,B 3.6599,C 0.053,E1 3.6506,E2 357.8183} C_DIS
LIN {X -15.9841,Y 138.189,Z 184,A 97.9614,B 3.6599,C 0.0526,E1 3.6437,E2 355.3392} C_DIS
LIN {X -20.9141,Y 137.5288,Z 184,A 100.0074,B 3.6599,C 0.0532,E1 3.638,E2 353.2946} C_DIS
LIN {X -25.7351,Y 136.7087,Z 184,A 101.9476,B 3.6599,C 0.0546,E1 3.6327,E2 351.3647} C_DIS
LIN {X -28.779,Y 136.1011,Z 184,A 103.2928,B 3.6599,C 0.0547,E1 3.629,E2 350.0118} C_DIS
LIN {X -33.0872,Y 135.118,Z 184,A 105.1396,B 3.6599,C 0.0556,E1 3.624,E2 348.1628} C_DIS
LIN {X -36.6135,Y 134.2068,Z 184,A 106.5072,B 3.6599,C 0.0575,E1 3.6204,E2 346.8126} C_DIS
LIN {X -40.4202,Y 133.1077,Z 184,A 108.1679,B 3.6599,C 0.0584,E1 3.6159,E2 345.1492} C_DIS
LIN {X -43.7292,Y 132.0575,Z 184,A 109.5897,B 3.6599,C 0.0596,E1 3.6121,E2 343.7292} C_DIS
LIN {X -48.4928,Y 130.3837,Z 184,A 111.881,B 3.6599,C 0.06,E1 3.606,E2 341.413} C_DIS
LIN {X -52.5033,Y 128.8217,Z 184,A 113.5293,B 3.6599,C 0.0625,E1 3.6018,E2 339.7813} C_DIS
LIN {X -56.3097,Y 127.2039,Z 184,A 115.2757,B 3.6599,C 0.064,E1 3.5973,E2 338.0307} C_DIS
LIN {X -59.2446,Y 125.8651,Z 184,A 116.7209,B 3.6598,C 0.0647,E1 3.5936,E2 336.5719} C_DIS
LIN {X -61.9097,Y 124.574,Z 184,A 118.1052,B 3.6598,C 0.0651,E1 3.5901,E2 335.1678} C_DIS
LIN {X -66.5866,Y 122.1397,Z 184,A 120.126,B 3.6598,C 0.0688,E1 3.5852,E2 333.1675} C_DIS
LIN {X -69.3122,Y 120.6147,Z 184,A 121.5354,B 3.6598,C 0.0697,E1 3.5817,E2 331.7437} C_DIS
LIN {X -73.4102,Y 118.1644,Z 184,A 123.4348,B 3.6596,C 0.0729,E1 3.5772,E2 329.854} C_DIS
LIN {X -76.6291,Y 116.1029,Z 184,A 125.0133,B 3.6596,C 0.0752,E1 3.5735,E2 328.2761} C_DIS
LIN {X -80.3195,Y 113.5812,Z 184,A 126.7049,B 3.6596,C 0.079,E1 3.5697,E2 326.6045} C_DIS
LIN {X -86.1401,Y 109.233,Z 184,A 129.7441,B 3.6594,C 0.0836,E1 3.5629,E2 323.5619} C_DIS
LIN {X -88.7601,Y 107.1146,Z 184,A 131.4324,B 3.6594,C 0.0842,E1 3.5592,E2 321.8372} C_DIS
LIN {X -92.3931,Y 103.9976,Z 184,A 133.9759,B 3.6594,C 0.0843,E1 3.5537,E2 319.2231} C_DIS
LIN {X -96.0771,Y 100.6036,Z 184,A 135.5035,B 3.6592,C 0.0914,E1 3.5507,E2 317.7646} C_DIS
LIN {X -98.8636,Y 97.8669,Z 184,A 137.2072,B 3.6592,C 0.094,E1 3.5473,E2 316.0503} C_DIS
LIN {X -102.027,Y 94.5647,Z 184,A 138.9066,B 3.659,C 0.0989,E1 3.5441,E2 314.3754} C_DIS
LIN {X -104.9691,Y 91.2876,Z 184,A 141.0447,B 3.659,C 0.1008,E1 3.5401,E2 312.1981} C_DIS
LIN {X -107.9339,Y 87.7626,Z 184,A 143.0355,B 3.6589,C 0.1043,E1 3.5365,E2 310.197} C_DIS
LIN {X -110.8287,Y 84.0774,Z 184,A 145.0073,B 3.6588,C 0.1084,E1 3.5331,E2 308.2215} C_DIS
LIN {X -113.3153,Y 80.6945,Z 184,A 147.0695,B 3.6588,C 0.1104,E1 3.5297,E2 306.1185} C_DIS
LIN {X -115.5054,Y 77.527,Z 184,A 148.7884,B 3.6586,C 0.1134,E1 3.527,E2 304.384} C_DIS
LIN {X -117.8525,Y 73.9111,Z 184,A 150.269,B 3.6584,C 0.1192,E1 3.5249,E2 302.9423} C_DIS
LIN {X -120.9395,Y 68.7429,Z 184,A 152.769,B 3.6582,C 0.1251,E1 3.5213,E2 300.4417} C_DIS
LIN {X -122.9591,Y 65.0582,Z 184,A 154.4393,B 3.6581,C 0.1297,E1 3.5191,E2 298.7803} C_DIS
LIN {X -124.6141,Y 61.8285,Z 184,A 156.0438,B 3.658,C 0.1329,E1 3.5171,E2 297.1631} C_DIS
LIN {X -126.1958,Y 58.5319,Z 184,A 157.6136,B 3.6578,C 0.1364,E1 3.5152,E2 295.5864} C_DIS
LIN {X -127.4712,Y 55.702,Z 184,A 158.8125,B 3.6577,C 0.1401,E1 3.5139,E2 294.3986} C_DIS
LIN {X -128.8472,Y 52.4401,Z 184,A 160.4985,B 3.6576,C 0.1427,E1 3.512,E2 292.6849} C_DIS
LIN {X -130.1864,Y 49.0195,Z 184,A 161.993,B 3.6574,C 0.1467,E1 3.5105,E2 291.1939} C_DIS
LIN {X -131.4023,Y 45.6597,Z 184,A 163.5458,B 3.6573,C 0.1502,E1 3.5091,E2 289.6319} C_DIS
LIN {X -132.4494,Y 42.5273,Z 184,A 164.9571,B 3.6571,C 0.1536,E1 3.5079,E2 288.2151} C_DIS
LIN {X -133.3363,Y 39.6632,Z 184,A 166.2226,B 3.6571,C 0.1568,E1 3.5068,E2 286.9467} C_DIS
LIN {X -134.3484,Y 36.0826,Z 184,A 167.8458,B 3.6569,C 0.1605,E1 3.5056,E2 285.3131} C_DIS
LIN {X -135.1557,Y 32.9311,Z 184,A 169.0778,B 3.6567,C 0.1647,E1 3.5048,E2 284.096} C_DIS
LIN {X -135.8758,Y 29.823,Z 184,A 170.6517,B 3.6566,C 0.167,E1 3.5038,E2 282.4898} C_DIS
LIN {X -136.6192,Y 26.2031,Z 184,A 172.2601,B 3.6564,C 0.1708,E1 3.5029,E2 280.8714} C_DIS
LIN {X -137.3545,Y 22.0396,Z 184,A 174.2167,B 3.6562,C 0.1746,E1 3.502,E2 278.8886} C_DIS
LIN {X -138.3236,Y 14.7666,Z 184,A 177.1594,B 3.6558,C 0.1834,E1 3.501,E2 275.9582} C_DIS
LIN {X -138.7105,Y 10.5374,Z 184,A 178.9115,B 3.6555,C 0.1884,E1 3.5006,E2 274.207} C_DIS
LIN {X -139.0363,Y 4.5528,Z 184,A -178.369,B 3.6552,C 0.1941,E1 3.5002,E2 271.4571} C_DIS
LIN {X -139.0989,Y -1.8034,Z 184,A -175.6615,B 3.6549,C 0.201,E1 3.5002,E2 268.7397} C_DIS
LIN {X -138.8269,Y -8.869,Z 184,A -172.6053,B 3.6544,C 0.2085,E1 3.5006,E2 265.6669} C_DIS
LIN {X -138.5912,Y -12.0004,Z 184,A -171.1981,B 3.6543,C 0.2115,E1 3.501,E2 264.2457} C_DIS
LIN {X -138.2295,Y -15.6412,Z 184,A -169.6719,B 3.654,C 0.2156,E1 3.5014,E2 262.718} C_DIS
LIN {X -137.7456,Y -19.4327,Z 184,A -168.1919,B 3.6537,C 0.2205,E1 3.502,E2 261.2512} C_DIS
LIN {X -137.1033,Y -23.549,Z 184,A -166.2583,B 3.6535,C 0.2242,E1 3.5028,E2 259.2903} C_DIS
LIN {X -136.3769,Y -27.4379,Z 184,A -164.6612,B 3.6532,C 0.2288,E1 3.5037,E2 257.6984} C_DIS
LIN {X -135.6416,Y -30.8668,Z 184,A -163.167,B 3.653,C 0.2325,E1 3.5046,E2 256.1984} C_DIS
LIN {X -134.8225,Y -34.268,Z 184,A -161.6003,B 3.6528,C 0.2358,E1 3.5057,E2 254.6161} C_DIS
LIN {X -133.6129,Y -38.7183,Z 184,A -159.6802,B 3.6524,C 0.2408,E1 3.5071,E2 252.6944} C_DIS
LIN {X -132.6437,Y -41.9189,Z 184,A -157.7343,B 3.6524,C 0.2414,E1 3.5088,E2 250.6744} C_DIS
LIN {X -131.1624,Y -46.351,Z 184,A -156.0145,B 3.652,C 0.2476,E1 3.5104,E2 248.9827} C_DIS
LIN {X -129.478,Y -50.863,Z 184,A -154.0778,B 3.6516,C 0.2531,E1 3.5123,E2 247.0531} C_DIS
LIN {X -127.6051,Y -55.3923,Z 184,A -152.0547,B 3.6513,C 0.2582,E1 3.5145,E2 245.0303} C_DIS
LIN {X -125.6852,Y -59.6213,Z 184,A -150.1175,B 3.6509,C 0.2629,E1 3.5168,E2 243.0907} C_DIS
LIN {X -124.1021,Y -62.8496,Z 184,A -148.6621,B 3.6506,C 0.2667,E1 3.5186,E2 241.6393} C_DIS
LIN {X -122.4901,Y -65.9399,Z 184,A -146.4776,B 3.6507,C 0.266,E1 3.5216,E2 239.3562} C_DIS
LIN {X -119.9748,Y -70.4127,Z 184,A -144.8431,B 3.6501,C 0.2738,E1 3.5238,E2 237.7862} C_DIS
LIN {X -117.2359,Y -74.8842,Z 184,A -142.6018,B 3.6498,C 0.2784,E1 3.5272,E2 235.5348} C_DIS
LIN {X -114.6898,Y -78.7282,Z 184,A -140.6884,B 3.6495,C 0.2827,E1 3.5301,E2 233.6201} C_DIS
LIN {X -112.868,Y -81.3194,Z 184,A -138.9854,B 3.6495,C 0.2832,E1 3.533,E2 231.8644} C_DIS
LIN {X -110.5693,Y -84.4175,Z 184,A -137.698,B 3.649,C 0.2885,E1 3.5351,E2 230.6177} C_DIS
LIN {X -107.9347,Y -87.7616,Z 184,A -135.8155,B 3.6488,C 0.2914,E1 3.5384,E2 228.7185} C_DIS
LIN {X -105.0052,Y -91.2462,Z 184,A -134.0124,B 3.6484,C 0.2958,E1 3.5417,E2 226.9253} C_DIS
LIN {X -102.2018,Y -94.3757,Z 184,A -132.1362,B 3.6482,C 0.2983,E1 3.5452,E2 225.03} C_DIS
LIN {X -99.2494,Y -97.4753,Z 184,A -130.1649,B 3.648,C 0.3005,E1 3.5491,E2 223.0312} C_DIS
LIN {X -95.5307,Y -101.1226,Z 184,A -128.1325,B 3.6476,C 0.3052,E1 3.5532,E2 221.0143} C_DIS
LIN {X -92.2391,Y -104.1338,Z 184,A -126.3355,B 3.6473,C 0.3088,E1 3.5569,E2 219.2229} C_DIS
LIN {X -89.3049,Y -106.6609,Z 184,A -124.618,B 3.6472,C 0.3107,E1 3.5606,E2 217.4892} C_DIS
LIN {X -85.6991,Y -109.5793,Z 184,A -122.7383,B 3.6469,C 0.3141,E1 3.5647,E2 215.6138} C_DIS
LIN {X -78.0342,Y -115.1632,Z 184,A -118.7541,B 3.6464,C 0.3196,E1 3.5738,E2 211.6194} C_DIS
LIN {X -74.3018,Y -117.6059,Z 184,A -116.7798,B 3.6463,C 0.3212,E1 3.5785,E2 209.6267} C_DIS
LIN {X -70.5838,Y -119.8742,Z 184,A -114.9535,B 3.6461,C 0.3234,E1 3.5828,E2 207.7959} C_DIS
LIN {X -66.0415,Y -122.4356,Z 184,A -111.7939,B 3.6465,C 0.3187,E1 3.591,E2 204.4989} C_DIS
LIN {X -59.3405,Y -125.8194,Z 184,A -109.7882,B 3.6455,C 0.3301,E1 3.5956,E2 202.6403} C_DIS
LIN {X -55.7224,Y -127.4624,Z 184,A -108.175,B 3.6453,C 0.332,E1 3.5997,E2 201.03} C_DIS
LIN {X -52.2636,Y -128.9183,Z 184,A -106.4734,B 3.6453,C 0.3323,E1 3.6042,E2 199.3072} C_DIS
LIN {X -48.4517,Y -130.3991,Z 184,A -104.5993,B 3.6453,C 0.3323,E1 3.6091,E2 197.4072} C_DIS
LIN {X -44.6848,Y -131.7392,Z 184,A -103.16,B 3.645,C 0.3352,E1 3.6129,E2 195.9956} C_DIS
LIN {X -42.1391,Y -132.5734,Z 184,A -101.9429,B 3.645,C 0.3351,E1 3.6161,E2 194.7629} C_DIS
LIN {X -37.854,Y -133.8604,Z 184,A -100.1635,B 3.6449,C 0.3368,E1 3.6209,E2 192.9915} C_DIS
LIN {X -34.2626,Y -134.8238,Z 184,A -97.8151,B 3.6454,C 0.3311,E1 3.6276,E2 190.5317} C_DIS
LIN {X -28.2931,Y -136.2029,Z 184,A -96.0267,B 3.6447,C 0.3382,E1 3.6322,E2 188.8426} C_DIS
LIN {X -23.7167,Y -137.0751,Z 184,A -93.9931,B 3.6447,C 0.3379,E1 3.6378,E2 186.7928} C_DIS
LIN {X -19.8981,Y -137.6791,Z 184,A -92.5721,B 3.6446,C 0.3398,E1 3.6417,E2 185.3944} C_DIS
LIN {X -16.4647,Y -138.1317,Z 184,A -91.1011,B 3.6446,C 0.3397,E1 3.6458,E2 183.9168} C_DIS
LIN {X -12.5162,Y -138.5475,Z 184,A -89.4054,B 3.6446,C 0.3394,E1 3.6505,E2 182.2123} C_DIS
LIN {X -9.3571,Y -138.7966,Z 184,A -88.0443,B 3.6446,C 0.339,E1 3.6543,E2 180.8431} C_DIS
LIN {X -5.6356,Y -138.9956,Z 184,A -86.6819,B 3.6446,C 0.3404,E1 3.6581,E2 179.5034} C_DIS
LIN {X -2.3662,Y -139.0895,Z 184,A -85.2786,B 3.6446,C 0.3398,E1 3.662,E2 178.0918} C_DIS
LIN {X 0.9893,Y -139.1038,Z 184,A -84.4225,B 3.6442,C 0.3442,E1 3.6642,E2 177.3059} C_DIS
Enddeposition()
LIN {X 0.9893,Y -139.1038,Z 184,A -84.4225,B 3.6442,C 0.3442,E1 3.6642,E2 177.3059} C_DIS
Startdeposition()
$VEL.CP = VEL_PRINT
LIN {X 0.0619,Y -140.0123,Z 184,A -85.0033,B 3.6251,C 0.3474,E1 3.6437,E2 177.9511} C_DIS
LIN {X -3.9745,Y -139.9541,Z 184,A -86.5244,B 3.6251,C 0.3464,E1 3.6395,E2 179.4551} C_DIS
LIN {X -8.1991,Y -139.7707,Z 184,A -88.2911,B 3.6251,C 0.3467,E1 3.6346,E2 181.2275} C_DIS
LIN {X -11.7612,Y -139.5155,Z 184,A -89.7352,B 3.6251,C 0.3465,E1 3.6305,E2 182.6699} C_DIS
LIN {X -15.1637,Y -139.1869,Z 184,A -91.0853,B 3.6252,C 0.3459,E1 3.6268,E2 184.0139} C_DIS
LIN {X -18.2378,Y -138.8174,Z 184,A -92.4025,B 3.6252,C 0.346,E1 3.6231,E2 185.3384} C_DIS
LIN {X -21.6758,Y -138.3224,Z 184,A -93.8258,B 3.6252,C 0.3457,E1 3.6192,E2 186.7625} C_DIS
LIN {X -25.9516,Y -137.5845,Z 184,A -95.6124,B 3.6253,C 0.3451,E1 3.6143,E2 188.5511} C_DIS
LIN {X -29.4997,Y -136.8671,Z 184,A -97.0653,B 3.6253,C 0.3443,E1 3.6103,E2 190.0007} C_DIS
LIN {X -33.7197,Y -135.891,Z 184,A -99.3221,B 3.6251,C 0.3472,E1 3.604,E2 192.3231} C_DIS
LIN {X -37.654,Y -134.8518,Z 184,A -100.256,B 3.6258,C 0.3405,E1 3.6018,E2 193.159} C_DIS
LIN {X -41.6322,Y -133.6789,Z 184,A -102.2135,B 3.6257,C 0.3414,E1 3.5964,E2 195.1523} C_DIS
LIN {X -49.359,Y -131.0212,Z 184,A -105.6547,B 3.6258,C 0.3395,E1 3.5873,E2 198.6073} C_DIS
LIN {X -52.7127,Y -129.7086,Z 184,A -107.1655,B 3.6259,C 0.3384,E1 3.5834,E2 200.1233} C_DIS
LIN {X -55.8492,Y -128.389,Z 184,A -108.6328,B 3.626,C 0.3376,E1 3.5796,E2 201.6009} C_DIS
LIN {X -60.1829,Y -126.4153,Z 184,A -110.519,B 3.6263,C 0.3351,E1 3.5748,E2 203.479} C_DIS
LIN {X -65.1287,Y -123.9396,Z 184,A -112.8573,B 3.6264,C 0.333,E1 3.569,E2 205.8275} C_DIS
LIN {X -67.6965,Y -122.5583,Z 184,A -114.1493,B 3.6265,C 0.3323,E1 3.5658,E2 207.133} C_DIS
LIN {X -71.5346,Y -120.3585,Z 184,A -115.9885,B 3.6267,C 0.3301,E1 3.5613,E2 208.9762} C_DIS
LIN {X -75.4744,Y -117.9278,Z 184,A -117.8576,B 3.627,C 0.3273,E1 3.5569,E2 210.8419} C_DIS
LIN {X -78.9531,Y -115.6281,Z 184,A -120.0642,B 3.6269,C 0.3282,E1 3.5516,E2 213.1152} C_DIS
LIN {X -82.5349,Y -113.0978,Z 184,A -121.6331,B 3.6273,C 0.3239,E1 3.5482,E2 214.654} C_DIS
LIN {X -86.8283,Y -109.8379,Z 184,A -123.7693,B 3.6276,C 0.3198,E1 3.5435,E2 216.7808} C_DIS
LIN {X -90.3827,Y -106.932,Z 184,A -125.815,B 3.6278,C 0.3177,E1 3.539,E2 218.8485} C_DIS
LIN {X -93.3472,Y -104.3535,Z 184,A -127.3305,B 3.6281,C 0.3143,E1 3.5359,E2 220.3516} C_DIS
LIN {X -99.5119,Y -98.4926,Z 184,A -130.7279,B 3.6287,C 0.3073,E1 3.5291,E2 223.7375} C_DIS
LIN {X -102.0941,Y -95.8137,Z 184,A -132.4505,B 3.6289,C 0.3055,E1 3.5257,E2 225.4864} C_DIS
LIN {X -106.2582,Y -91.1734,Z 184,A -135.063,B 3.6293,C 0.3007,E1 3.5208,E2 228.1064} C_DIS
LIN {X -109.1444,Y -87.6978,Z 184,A -137.9578,B 3.6291,C 0.3029,E1 3.5156,E2 231.1382} C_DIS
LIN {X -113.6372,Y -81.7931,Z 184,A -140.1561,B 3.63,C 0.2913,E1 3.5121,E2 233.2259} C_DIS
LIN {X -116.2268,Y -78.0693,Z 184,A -142.0796,B 3.6303,C 0.2875,E1 3.509,E2 235.1578} C_DIS
LIN {X -118.7669,Y -74.147,Z 184,A -143.8268,B 3.6308,C 0.2821,E1 3.5064,E2 236.8825} C_DIS
LIN {X -120.3132,Y -71.6106,Z 184,A -145.4664,B 3.6308,C 0.2816,E1 3.504,E2 238.5776} C_DIS
LIN {X -121.9273,Y -68.8255,Z 184,A -146.7973,B 3.631,C 0.2785,E1 3.5022,E2 239.9098} C_DIS
LIN {X -124.3339,Y -64.3778,Z 184,A -148.6807,B 3.6315,C 0.2724,E1 3.4997,E2 241.7679} C_DIS
LIN {X -125.697,Y -61.6694,Z 184,A -149.9812,B 3.6317,C 0.2697,E1 3.4981,E2 243.0757} C_DIS
LIN {X -127.1745,Y -58.5617,Z 184,A -151.4282,B 3.6319,C 0.2663,E1 3.4964,E2 244.5271} C_DIS
LIN {X -128.9558,Y -54.5304,Z 184,A -153.2105,B 3.6323,C 0.2616,E1 3.4944,E2 246.3059} C_DIS
LIN {X -129.8716,Y -52.3081,Z 184,A -154.8685,B 3.6323,C 0.2627,E1 3.4926,E2 248.0515} C_DIS
LIN {X -131.5437,Y -47.9504,Z 184,A -156.7605,B 3.6326,C 0.2576,E1 3.4908,E2 249.9402} C_DIS
LIN {X -132.8905,Y -44.0787,Z 184,A -158.0112,B 3.633,C 0.2509,E1 3.4897,E2 251.1345} C_DIS
LIN {X -133.7982,Y -41.2425,Z 184,A -159.3749,B 3.6332,C 0.2484,E1 3.4886,E2 252.5166} C_DIS
LIN {X -134.8343,Y -37.7164,Z 184,A -160.8656,B 3.6335,C 0.2443,E1 3.4874,E2 254.0047} C_DIS
LIN {X -135.7105,Y -34.431,Z 184,A -162.3405,B 3.6337,C 0.2409,E1 3.4864,E2 255.4897} C_DIS
LIN {X -136.536,Y -30.9968,Z 184,A -163.8402,B 3.634,C 0.2372,E1 3.4854,E2 256.9957} C_DIS
LIN {X -137.3391,Y -27.227,Z 184,A -165.4977,B 3.6342,C 0.2333,E1 3.4845,E2 258.6627} C_DIS
LIN {X -138.5617,Y -20.0898,Z 184,A -168.3317,B 3.6348,C 0.2244,E1 3.4832,E2 261.4783} C_DIS
LIN {X -139.015,Y -16.6653,Z 184,A -170.6609,B 3.6348,C 0.2251,E1 3.4824,E2 263.9248} C_DIS
LIN {X -139.5307,Y -11.5818,Z 184,A -171.7942,B 3.6354,C 0.2144,E1 3.4821,E2 264.9332} C_DIS
LIN {X -139.9318,Y -4.7454,Z 184,A -175.0556,B 3.6357,C 0.2089,E1 3.4816,E2 268.2525} C_DIS
LIN {X -139.9872,Y 2.5615,Z 184,A -178.116,B 3.6362,C 0.2008,E1 3.4816,E2 271.32} C_DIS
LIN {X -139.6339,Y 10.2607,Z 184,A 177.9852,B 3.6364,C 0.1956,E1 3.4822,E2 275.312} C_DIS
LIN {X -139.244,Y 14.6326,Z 184,A 176.2299,B 3.6367,C 0.1904,E1 3.4827,E2 277.0609} C_DIS
LIN {X -138.8045,Y 18.3362,Z 184,A 174.6069,B 3.6369,C 0.1866,E1 3.4833,E2 278.695} C_DIS
LIN {X -138.2171,Y 22.3469,Z 184,A 173.3606,B 3.6372,C 0.1799,E1 3.4838,E2 279.8876} C_DIS
LIN {X -137.4728,Y 26.5359,Z 184,A 171.5015,B 3.6375,C 0.1756,E1 3.4847,E2 281.7604} C_DIS
LIN {X -136.349,Y 31.8153,Z 184,A 169.2178,B 3.6377,C 0.1699,E1 3.4861,E2 284.0521} C_DIS
LIN {X -135.4542,Y 35.4321,Z 184,A 167.5213,B 3.6379,C 0.1666,E1 3.4873,E2 285.7693} C_DIS
LIN {X -134.3608,Y 39.37,Z 184,A 165.8762,B 3.6381,C 0.1619,E1 3.4885,E2 287.4095} C_DIS
LIN {X -133.3679,Y 42.6122,Z 184,A 164.4236,B 3.6382,C 0.1585,E1 3.4897,E2 288.8694} C_DIS
LIN {X -132.2503,Y 45.9638,Z 184,A 162.9036,B 3.6384,C 0.155,E1 3.4911,E2 290.3977} C_DIS
LIN {X -130.9665,Y 49.505,Z 184,A 161.3414,B 3.6386,C 0.1511,E1 3.4926,E2 291.9613} C_DIS
LIN {X -129.6844,Y 52.7727,Z 184,A 159.8365,B 3.6386,C 0.1477,E1 3.4942,E2 293.4737} C_DIS
LIN {X -128.2194,Y 56.2416,Z 184,A 158.2473,B 3.6388,C 0.1439,E1 3.4959,E2 295.0678} C_DIS
LIN {X -127.0142,Y 58.9084,Z 184,A 156.9486,B 3.6389,C 0.1414,E1 3.4975,E2 296.3784} C_DIS
LIN {X -125.4166,Y 62.2378,Z 184,A 155.4179,B 3.6391,C 0.1377,E1 3.4993,E2 297.9103} C_DIS
LIN {X -123.7586,Y 65.4733,Z 184,A 153.8576,B 3.6392,C 0.1343,E1 3.5014,E2 299.4786} C_DIS
LIN {X -121.632,Y 69.3469,Z 184,A 151.9648,B 3.6394,C 0.1304,E1 3.5039,E2 301.3806} C_DIS
LIN {X -120.227,Y 71.7553,Z 184,A 150.7349,B 3.6394,C 0.1281,E1 3.5057,E2 302.6208} C_DIS
LIN {X -116.5277,Y 77.6184,Z 184,A 147.783,B 3.6396,C 0.122,E1 3.5102,E2 305.5849} C_DIS
LIN {X -114.4718,Y 80.6198,Z 184,A 146.4505,B 3.6398,C 0.1177,E1 3.5123,E2 306.8966} C_DIS
LIN {X -112.4069,Y 83.4749,Z 184,A 144.7655,B 3.6398,C 0.1158,E1 3.5151,E2 308.6109} C_DIS
LIN {X -109.7267,Y 86.9682,Z 184,A 142.6021,B 3.6399,C 0.1139,E1 3.5189,E2 310.8181} C_DIS
LIN {X -107.2968,Y 89.9485,Z 184,A 140.5336,B 3.6399,C 0.1133,E1 3.5228,E2 312.9464} C_DIS
LIN {X -103.1823,Y 94.6402,Z 184,A 139.0185,B 3.6403,C 0.1022,E1 3.5253,E2 314.3305} C_DIS
LIN {X -101.2406,Y 96.7144,Z 184,A 137.462,B 3.6403,C 0.1021,E1 3.5284,E2 315.9354} C_DIS
LIN {X -98.0612,Y 99.9366,Z 184,A 135.5545,B 3.6403,C 0.0988,E1 3.5322,E2 317.8484} C_DIS
LIN {X -94.1179,Y 103.6589,Z 184,A 133.3244,B 3.6405,C 0.0947,E1 3.5367,E2 320.0781} C_DIS
LIN {X -90.9376,Y 106.4603,Z 184,A 131.4578,B 3.6405,C 0.0923,E1 3.5407,E2 321.9598} C_DIS
LIN {X -87.594,Y 109.228,Z 184,A 129.6548,B 3.6405,C 0.0894,E1 3.5446,E2 323.7648} C_DIS
LIN {X -83.1646,Y 112.637,Z 184,A 127.3852,B 3.6407,C 0.0855,E1 3.5497,E2 326.0306} C_DIS
LIN {X -80.8139,Y 114.3349,Z 184,A 126.1085,B 3.6407,C 0.0842,E1 3.5526,E2 327.3176} C_DIS
LIN {X -76.1565,Y 117.4885,Z 184,A 123.8123,B 3.6407,C 0.0807,E1 3.5579,E2 329.6114} C_DIS
LIN {X -69.7603,Y 121.3962,Z 184,A 120.7681,B 3.6409,C 0.0763,E1 3.5652,E2 332.6506} C_DIS
LIN {X -66.544,Y 123.1882,Z 184,A 119.0645,B 3.6409,C 0.0757,E1 3.5694,E2 334.3776} C_DIS
LIN {X -59.1495,Y 126.9027,Z 184,A 115.9198,B 3.641,C 0.0701,E1 3.5773,E2 337.4901} C_DIS
LIN {X -55.2135,Y 128.6639,Z 184,A 113.6136,B 3.641,C 0.0718,E1 3.5833,E2 339.862} C_DIS
LIN {X -51.8081,Y 130.0732,Z 184,A 112.5045,B 3.641,C 0.0677,E1 3.5861,E2 340.921} C_DIS
LIN {X -46.2159,Y 132.1629,Z 184,A 110.1435,B 3.6411,C 0.0649,E1 3.5922,E2 343.2704} C_DIS
LIN {X -42.2875,Y 133.4717,Z 184,A 108.2435,B 3.6411,C 0.065,E1 3.5973,E2 345.1948} C_DIS
LIN {X -38.7046,Y 134.5556,Z 184,A 106.3567,B 3.6411,C 0.0664,E1 3.6025,E2 347.1244} C_DIS
LIN {X -35.1865,Y 135.5188,Z 184,A 105.2309,B 3.6411,C 0.0629,E1 3.6054,E2 348.2042} C_DIS
LIN {X -30.7499,Y 136.5924,Z 184,A 103.3259,B 3.6411,C 0.0621,E1 3.6106,E2 350.1126} C_DIS
LIN {X -27.0011,Y 137.3838,Z 184,A 101.7856,B 3.6411,C 0.0611,E1 3.6148,E2 351.6488} C_DIS
LIN {X -19.3579,Y 138.6663,Z 184,A 98.5688,B 3.6411,C 0.0604,E1 3.6237,E2 354.8695} C_DIS
LIN {X -15.4705,Y 139.1539,Z 184,A 96.7615,B 3.6411,C 0.0615,E1 3.6288,E2 356.7013} C_DIS
LIN {X -9.2656,Y 139.705,Z 184,A 94.4486,B 3.6412,C 0.0594,E1 3.6351,E2 358.9838} C_DIS
LIN {X -5.4844,Y 139.903,Z 184,A 92.8322,B 3.6412,C 0.0598,E1 3.6397,E2 360.6077} C_DIS
LIN {X -1.9148,Y 139.998,Z 184,A 91.3865,B 3.6412,C 0.0598,E1 3.6437,E2 362.0508} C_DIS
LIN {X 2.0179,Y 139.9963,Z 184,A 89.6656,B 3.6412,C 0.0608,E1 3.6486,E2 363.7848} C_DIS
LIN {X 5.5682,Y 139.8997,Z 184,A 88.3049,B 3.6412,C 0.0604,E1 3.6523,E2 365.1335} C_DIS
LIN {X 9.392,Y 139.6972,Z 184,A 86.6101,B 3.6412,C 0.0618,E1 3.6571,E2 366.8436} C_DIS
LIN {X 13.4269,Y 139.3651,Z 184,A 85.0814,B 3.6412,C 0.0613,E1 3.6613,E2 368.3558} C_DIS
LIN {X 16.9172,Y 138.9849,Z 184,A 83.6791,B 3.6412,C 0.0616,E1 3.6652,E2 369.7533} C_DIS
LIN {X 20.9581,Y 138.4336,Z 184,A 81.9013,B 3.6412,C 0.0634,E1 3.6701,E2 371.544} C_DIS
LIN {X 24.7743,Y 137.801,Z 184,A 80.4414,B 3.6412,C 0.0632,E1 3.6741,E2 372.9882} C_DIS
LIN {X 28.156,Y 137.1501,Z 184,A 78.8792,B 3.6411,C 0.0655,E1 3.6784,E2 374.5688} C_DIS
LIN {X 34.4395,Y 135.7083,Z 184,A 76.7505,B 3.6411,C 0.063,E1 3.6841,E2 376.6336} C_DIS
LIN {X 37.7932,Y 134.8128,Z 184,A 75.0329,B 3.6411,C 0.0668,E1 3.6888,E2 378.3879} C_DIS
LIN {X 41.1168,Y 133.8366,Z 184,A 73.0005,B 3.6409,C 0.0735,E1 3.6944,E2 380.4958} C_DIS
LIN {X 46.1373,Y 132.1902,Z 184,A 71.4911,B 3.641,C 0.0698,E1 3.6982,E2 381.9244} C_DIS
LIN {X 49.2067,Y 131.0783,Z 184,A 70.1885,B 3.641,C 0.0709,E1 3.7016,E2 383.2225} C_DIS
LIN {X 52.6808,Y 129.7215,Z 184,A 68.7314,B 3.641,C 0.072,E1 3.7054,E2 384.6708} C_DIS
LIN {X 55.8823,Y 128.3747,Z 184,A 67.2693,B 3.641,C 0.0741,E1 3.7091,E2 386.1377} C_DIS
LIN {X 59.4472,Y 126.765,Z 184,A 65.3516,B 3.6408,C 0.0791,E1 3.7141,E2 388.0947} C_DIS
LIN {X 62.7766,Y 125.1488,Z 184,A 64.2719,B 3.6408,C 0.077,E1 3.7167,E2 389.1202} C_DIS
LIN {X 66.3708,Y 123.2813,Z 184,A 62.5114,B 3.6408,C 0.0803,E1 3.7211,E2 390.8935} C_DIS
LIN {X 70.3818,Y 121.0364,Z 184,A 60.6971,B 3.6408,C 0.0824,E1 3.7254,E2 392.6994} C_DIS
LIN {X 73.9322,Y 118.9006,Z 184,A 59.0063,B 3.6407,C 0.0849,E1 3.7295,E2 394.3896} C_DIS
LIN {X 77.6868,Y 116.4822,Z 184,A 56.9243,B 3.6406,C 0.0904,E1 3.7344,E2 396.5032} C_DIS
LIN {X 80.9076,Y 114.2687,Z 184,A 55.6407,B 3.6406,C 0.09,E1 3.7372,E2 397.7476} C_DIS
LIN {X 84.6563,Y 111.5204,Z 184,A 53.7821,B 3.6406,C 0.0929,E1 3.7414,E2 399.6008} C_DIS
LIN {X 88.221,Y 108.7223,Z 184,A 52.018,B 3.6404,C 0.0953,E1 3.7452,E2 401.3537} C_DIS
LIN {X 90.6603,Y 106.696,Z 184,A 50.903,B 3.6404,C 0.0959,E1 3.7476,E2 402.4459} C_DIS
LIN {X 94.3438,Y 103.4536,Z 184,A 48.6165,B 3.6402,C 0.1026,E1 3.7524,E2 404.7676} C_DIS
LIN {X 98,Y 99.9967,Z 184,A 46.7597,B 3.6402,C 0.1047,E1 3.7561,E2 406.5993} C_DIS
LIN {X 101.2804,Y 96.6728,Z 184,A 44.9204,B 3.6401,C 0.1079,E1 3.7596,E2 408.4299} C_DIS
LIN {X 104.2909,Y 93.4171,Z 184,A 43.173,B 3.64,C 0.111,E1 3.7629,E2 410.1692} C_DIS
LIN {X 107.1363,Y 90.1398,Z 184,A 41.1074,B 3.6398,C 0.1179,E1 3.7667,E2 412.2717} C_DIS
LIN {X 109.6762,Y 87.0312,Z 184,A 39.8069,B 3.6398,C 0.118,E1 3.7689,E2 413.5295} C_DIS
LIN {X 112.0927,Y 83.8968,Z 184,A 38.2263,B 3.6397,C 0.1213,E1 3.7716,E2 415.1056} C_DIS
LIN {X 114.7948,Y 80.1595,Z 184,A 36.4312,B 3.6396,C 0.1247,E1 3.7745,E2 416.8895} C_DIS
LIN {X 117.2845,Y 76.4706,Z 184,A 34.6549,B 3.6394,C 0.1286,E1 3.7772,E2 418.6607} C_DIS
LIN {X 119.6518,Y 72.711,Z 184,A 32.8817,B 3.6393,C 0.1325,E1 3.7798,E2 420.4289} C_DIS
LIN {X 122.0022,Y 68.6936,Z 184,A 31.0681,B 3.6391,C 0.1362,E1 3.7823,E2 422.2316} C_DIS
LIN {X 124.0939,Y 64.8347,Z 184,A 29.4177,B 3.6391,C 0.1391,E1 3.7845,E2 423.864} C_DIS
LIN {X 125.7977,Y 61.4653,Z 184,A 27.9452,B 3.6389,C 0.1423,E1 3.7863,E2 425.3279} C_DIS
LIN {X 127.2545,Y 58.3886,Z 184,A 26.5996,B 3.6388,C 0.1453,E1 3.7879,E2 426.668} C_DIS
LIN {X 128.5844,Y 55.3973,Z 184,A 25.2919,B 3.6387,C 0.1484,E1 3.7893,E2 427.9721} C_DIS
LIN {X 129.953,Y 52.1064,Z 184,A 23.8359,B 3.6385,C 0.1522,E1 3.7909,E2 429.4285} C_DIS
LIN {X 131.4625,Y 48.1762,Z 184,A 22.2359,B 3.6384,C 0.1555,E1 3.7924,E2 431.0136} C_DIS
LIN {X 132.7244,Y 44.5777,Z 184,A 20.6807,B 3.6382,C 0.1596,E1 3.7938,E2 432.5688} C_DIS
LIN {X 133.9,Y 40.9096,Z 184,A 19.1358,B 3.638,C 0.1635,E1 3.7951,E2 434.1105} C_DIS
LIN {X 135.5558,Y 35.0406,Z 184,A 16.8806,B 3.6378,C 0.1676,E1 3.7968,E2 436.3362} C_DIS
LIN {X 136.6126,Y 30.6614,Z 184,A 14.6079,B 3.6374,C 0.1775,E1 3.7982,E2 438.6651} C_DIS
LIN {X 137.4449,Y 26.6815,Z 184,A 12.8491,B 3.6371,C 0.1832,E1 3.7992,E2 440.437} C_DIS
LIN {X 138.3082,Y 21.7678,Z 184,A 11.4477,B 3.6371,C 0.1817,E1 3.7998,E2 441.7573} C_DIS
LIN {X 138.8071,Y 18.3159,Z 184,A 10.0509,B 3.637,C 0.1853,E1 3.8003,E2 443.151} C_DIS
LIN {X 139.1779,Y 15.2473,Z 184,A 8.8547,B 3.6368,C 0.1881,E1 3.8007,E2 444.3391} C_DIS
LIN {X 139.5223,Y 11.6803,Z 184,A 7.4092,B 3.6366,C 0.192,E1 3.801,E2 445.7828} C_DIS
LIN {X 139.8008,Y 7.6874,Z 184,A 5.7844,B 3.6364,C 0.1964,E1 3.8013,E2 447.4071} C_DIS
LIN {X 139.9579,Y 3.8348,Z 184,A 4.3361,B 3.6362,C 0.1994,E1 3.8015,E2 448.8395} C_DIS
LIN {X 140.0097,Y -0.5025,Z 184,A 2.6401,B 3.636,C 0.2035,E1 3.8015,E2 450.5264} C_DIS
LIN {X 139.9487,Y -4.1684,Z 184,A 1.2025,B 3.6358,C 0.2071,E1 3.8014,E2 451.9569} C_DIS
LIN {X 139.7792,Y -8.0617,Z 184,A -0.4016,B 3.6355,C 0.2117,E1 3.8012,E2 453.5633} C_DIS
LIN {X 139.5133,Y -11.7876,Z 184,A -1.8276,B 3.6354,C 0.2148,E1 3.8009,E2 454.9769} C_DIS
LIN {X 139.1851,Y -15.1803,Z 184,A -3.1201,B 3.6352,C 0.2176,E1 3.8005,E2 456.2571} C_DIS
LIN {X 138.7666,Y -18.6251,Z 184,A -4.4998,B 3.635,C 0.2211,E1 3.8,E2 457.6325} C_DIS
LIN {X 138.2272,Y -22.2864,Z 184,A -5.9364,B 3.6348,C 0.2245,E1 3.7994,E2 459.0601} C_DIS
LIN {X 137.7011,Y -25.3323,Z 184,A -7.7854,B 3.6341,C 0.2346,E1 3.7984,E2 460.9863} C_DIS
LIN {X 136.6671,Y -30.4227,Z 184,A -9.2037,B 3.6343,C 0.2325,E1 3.7977,E2 462.3139} C_DIS
LIN {X 135.1074,Y -36.7326,Z 184,A -11.7701,B 3.6339,C 0.2388,E1 3.7959,E2 464.8702} C_DIS
LIN {X 134.2202,Y -39.8502,Z 184,A -13.0637,B 3.6336,C 0.242,E1 3.7949,E2 466.1605} C_DIS
LIN {X 133.1177,Y -43.3952,Z 184,A -14.7362,B 3.6333,C 0.2479,E1 3.7935,E2 467.8544} C_DIS
LIN {X 130.8557,Y -49.8007,Z 184,A -17.2009,B 3.633,C 0.2518,E1 3.7912,E2 470.2797} C_DIS
LIN {X 129.7087,Y -52.7125,Z 184,A -18.4837,B 3.6327,C 0.2552,E1 3.7898,E2 471.5638} C_DIS
LIN {X 128.1028,Y -56.5064,Z 184,A -20.4874,B 3.6322,C 0.2632,E1 3.7875,E2 473.6108} C_DIS
LIN {X 126.4557,Y -60.0984,Z 184,A -21.4408,B 3.6324,C 0.2599,E1 3.7865,E2 474.4778} C_DIS
LIN {X 125.2776,Y -62.5195,Z 184,A -22.7219,B 3.6321,C 0.2647,E1 3.7849,E2 475.7835} C_DIS
LIN {X 122.0863,Y -68.544,Z 184,A -25.4998,B 3.6316,C 0.2717,E1 3.7812,E2 478.5622} C_DIS
LIN {X 119.7392,Y -72.5663,Z 184,A -27.3305,B 3.6313,C 0.2755,E1 3.7786,E2 480.3846} C_DIS
LIN {X 117.3583,Y -76.3569,Z 184,A -29.1975,B 3.6309,C 0.2804,E1 3.7758,E2 482.2578} C_DIS
LIN {X 115.3557,Y -79.35,Z 184,A -30.6007,B 3.6307,C 0.2831,E1 3.7736,E2 483.6528} C_DIS
LIN {X 111.362,Y -84.864,Z 184,A -32.9247,B 3.6306,C 0.2845,E1 3.7699,E2 485.9175} C_DIS
LIN {X 108.1658,Y -88.9024,Z 184,A -35.2605,B 3.63,C 0.2918,E1 3.7657,E2 488.2856} C_DIS
LIN {X 103.6576,Y -94.1192,Z 184,A -37.9945,B 3.6296,C 0.2971,E1 3.7607,E2 491.0103} C_DIS
LIN {X 100.554,Y -97.4281,Z 184,A -39.8179,B 3.6293,C 0.3006,E1 3.7572,E2 492.8308} C_DIS
LIN {X 95.8584,Y -102.0519,Z 184,A -42.8528,B 3.6285,C 0.3097,E1 3.751,E2 495.9129} C_DIS
LIN {X 92.4376,Y -105.1607,Z 184,A -44.2982,B 3.6285,C 0.3087,E1 3.7481,E2 497.3004} C_DIS
LIN {X 89.0804,Y -108.0189,Z 184,A -46.5698,B 3.6279,C 0.3171,E1 3.7431,E2 499.6357} C_DIS
LIN {X 84.9571,Y -111.2908,Z 184,A -48.3902,B 3.6279,C 0.3175,E1 3.7392,E2 501.4134} C_DIS
LIN {X 81.9979,Y -113.4888,Z 184,A -49.5405,B 3.6279,C 0.3164,E1 3.7367,E2 502.5169} C_DIS
LIN {X 78.5592,Y -115.8956,Z 184,A -51.2546,B 3.6277,C 0.3193,E1 3.7327,E2 504.2318} C_DIS
LIN {X 72.1342,Y -120.0006,Z 184,A -54.2759,B 3.6273,C 0.3234,E1 3.7256,E2 507.2424} C_DIS
LIN {X 68.5611,Y -122.0767,Z 184,A -55.9753,B 3.6271,C 0.326,E1 3.7215,E2 508.9441} C_DIS
LIN {X 64.68,Y -124.1752,Z 184,A -57.7129,B 3.6269,C 0.3279,E1 3.7172,E2 510.6738} C_DIS
LIN {X 60.1148,Y -126.4478,Z 184,A -59.7018,B 3.6267,C 0.3298,E1 3.7122,E2 512.6511} C_DIS
LIN {X 55.1229,Y -128.7031,Z 184,A -61.9992,B 3.6264,C 0.3332,E1 3.7064,E2 514.9576} C_DIS
LIN {X 51.0644,Y -130.3662,Z 184,A -64.1196,B 3.6259,C 0.3385,E1 3.7007,E2 517.123} C_DIS
LIN {X 47.1965,Y -131.8157,Z 184,A -65.358,B 3.6262,C 0.336,E1 3.6976,E2 518.3018} C_DIS
LIN {X 44.0445,Y -132.902,Z 184,A -66.7,B 3.6261,C 0.3372,E1 3.6941,E2 519.6417} C_DIS
LIN {X 40.6703,Y -133.9733,Z 184,A -68.1562,B 3.6259,C 0.3386,E1 3.6902,E2 521.0998} C_DIS
LIN {X 36.8451,Y -135.0773,Z 184,A -69.9408,B 3.6257,C 0.3416,E1 3.6853,E2 522.9065} C_DIS
LIN {X 32.0807,Y -136.2873,Z 184,A -71.71,B 3.6257,C 0.3409,E1 3.6806,E2 524.6443} C_DIS
LIN {X 28.6922,Y -137.041,Z 184,A -73.6788,B 3.6251,C 0.3471,E1 3.675,E2 526.6877} C_DIS
LIN {X 24.0524,Y -137.9302,Z 184,A -75.0798,B 3.6255,C 0.3434,E1 3.6714,E2 528.0183} C_DIS
LIN {X 19.1843,Y -138.6911,Z 184,A -77.032,B 3.6255,C 0.344,E1 3.666,E2 529.963} C_DIS
LIN {X 15.7012,Y -139.129,Z 184,A -78.5878,B 3.6253,C 0.3458,E1 3.6616,E2 531.5357} C_DIS
LIN {X 11.837,Y -139.5091,Z 184,A -80.0821,B 3.6253,C 0.3455,E1 3.6575,E2 533.0179} C_DIS
LIN {X 7.5836,Y -139.806,Z 184,A -81.8346,B 3.6253,C 0.3462,E1 3.6526,E2 534.7725} C_DIS
LIN {X 3.9013,Y -139.9561,Z 184,A -83.2833,B 3.6253,C 0.346,E1 3.6486,E2 536.2139} C_DIS
LIN {X 0.9975,Y -140.0038,Z 184,A -84.0745,B 3.6255,C 0.3428,E1 3.6465,E2 536.9516} C_DIS
Enddeposition()
LIN {X 0.9975,Y -140.0038,Z 184,A -84.0745,B 3.6255,C 0.3428,E1 3.6465,E2 536.9516} C_DIS
Startdeposition()
$VEL.CP = VEL_PRINT
LIN {X 3.4946,Y -140.8686,Z 184,A -82.6741,B 3.5602,C 0.339,E1 3.585,E2 535.5477} C_DIS
LIN {X 7.483,Y -140.713,Z 184,A -81.0307,B 3.5602,C 0.3384,E1 3.5895,E2 533.9007} C_DIS
LIN {X 11.7,Y -140.4247,Z 184,A -79.4131,B 3.5602,C 0.3387,E1 3.594,E2 532.2961} C_DIS
LIN {X 15.8758,Y -140.0163,Z 184,A -77.6697,B 3.5603,C 0.3376,E1 3.5989,E2 530.5467} C_DIS
LIN {X 23.4575,Y -138.9451,Z 184,A -74.6231,B 3.5604,C 0.3364,E1 3.6073,E2 527.5076} C_DIS
LIN {X 27.7228,Y -138.1576,Z 184,A -72.9513,B 3.5604,C 0.3361,E1 3.6118,E2 525.8474} C_DIS
LIN {X 31.1093,Y -137.4343,Z 184,A -71.5686,B 3.5605,C 0.3353,E1 3.6156,E2 524.4674} C_DIS
LIN {X 34.123,Y -136.7181,Z 184,A -70.3819,B 3.5605,C 0.3349,E1 3.6188,E2 523.29} C_DIS
LIN {X 38.2083,Y -135.6322,Z 184,A -68.5532,B 3.5608,C 0.3324,E1 3.6238,E2 521.445} C_DIS
LIN {X 42.2156,Y -134.4404,Z 184,A -66.8083,B 3.561,C 0.3303,E1 3.6284,E2 519.6928} C_DIS
LIN {X 45.2897,Y -133.4368,Z 184,A -65.2385,B 3.5613,C 0.3265,E1 3.6327,E2 518.087} C_DIS
LIN {X 48.8115,Y -132.1882,Z 184,A -64.0292,B 3.5613,C 0.3278,E1 3.6358,E2 516.9194} C_DIS
LIN {X 52.2031,Y -130.8853,Z 184,A -62.7267,B 3.5613,C 0.3278,E1 3.6391,E2 515.6399} C_DIS
LIN {X 55.9417,Y -129.3305,Z 184,A -60.3097,B 3.5621,C 0.3181,E1 3.6456,E2 513.1154} C_DIS
LIN {X 61.345,Y -126.8584,Z 184,A -58.5718,B 3.5618,C 0.3217,E1 3.6497,E2 511.4696} C_DIS
LIN {X 64.8269,Y -125.1155,Z 184,A -56.9917,B 3.562,C 0.3195,E1 3.6537,E2 509.8888} C_DIS
LIN {X 68.7802,Y -122.9869,Z 184,A -55.2072,B 3.5622,C 0.3172,E1 3.658,E2 508.1086} C_DIS
LIN {X 71.7899,Y -121.2551,Z 184,A -53.9686,B 3.5622,C 0.3168,E1 3.6609,E2 506.8927} C_DIS
LIN {X 75.0059,Y -119.2913,Z 184,A -51.9581,B 3.5629,C 0.3094,E1 3.6659,E2 504.8151} C_DIS
LIN {X 78.8078,Y -116.8152,Z 184,A -50.5393,B 3.5627,C 0.3107,E1 3.669,E2 503.4536} C_DIS
LIN {X 81.5548,Y -114.9147,Z 184,A -48.6562,B 3.5634,C 0.3029,E1 3.6735,E2 501.4973} C_DIS
LIN {X 85.9827,Y -111.6404,Z 184,A -46.1521,B 3.564,C 0.296,E1 3.6791,E2 498.9546} C_DIS
LIN {X 91.684,Y -107.0074,Z 184,A -44.393,B 3.5634,C 0.3034,E1 3.6825,E2 497.3623} C_DIS
LIN {X 94.9002,Y -104.164,Z 184,A -42.2975,B 3.564,C 0.2962,E1 3.687,E2 495.2176} C_DIS
LIN {X 101.2807,Y -97.9726,Z 184,A -38.9378,B 3.5644,C 0.2915,E1 3.6936,E2 491.89} C_DIS
LIN {X 103.2818,Y -95.861,Z 184,A -37.6129,B 3.5647,C 0.2874,E1 3.6961,E2 490.5448} C_DIS
LIN {X 108.0436,Y -90.4599,Z 184,A -34.9625,B 3.565,C 0.284,E1 3.7009,E2 487.9299} C_DIS
LIN {X 110.8222,Y -87.0336,Z 184,A -33.2442,B 3.5652,C 0.2807,E1 3.7039,E2 486.2204} C_DIS
LIN {X 114.4885,Y -82.1514,Z 184,A -30.7656,B 3.5657,C 0.275,E1 3.708,E2 483.7403} C_DIS
LIN {X 116.627,Y -79.0857,Z 184,A -29.3036,B 3.5659,C 0.272,E1 3.7103,E2 482.2849} C_DIS
LIN {X 119.1952,Y -75.1592,Z 184,A -27.4939,B 3.5662,C 0.2685,E1 3.713,E2 480.4869} C_DIS
LIN {X 121.5777,Y -71.2412,Z 184,A -25.8574,B 3.5663,C 0.2664,E1 3.7153,E2 478.8797} C_DIS
LIN {X 126.4299,Y -62.2201,Z 184,A -22.0801,B 3.5668,C 0.2603,E1 3.7203,E2 475.1518} C_DIS
LIN {X 128.6823,Y -57.417,Z 184,A -19.6477,B 3.5674,C 0.2516,E1 3.7232,E2 472.6806} C_DIS
LIN {X 130.0283,Y -54.3,Z 184,A -18.3076,B 3.5676,C 0.2484,E1 3.7246,E2 471.3448} C_DIS
LIN {X 131.3104,Y -51.1218,Z 184,A -17.1537,B 3.5676,C 0.2474,E1 3.7258,E2 470.2221} C_DIS
LIN {X 133.6173,Y -44.7476,Z 184,A -14.5399,B 3.5681,C 0.2417,E1 3.7282,E2 467.6253} C_DIS
LIN {X 134.9597,Y -40.5256,Z 184,A -12.4671,B 3.5686,C 0.2337,E1 3.73,E2 465.5148} C_DIS
LIN {X 135.7775,Y -37.6887,Z 184,A -11.2387,B 3.5688,C 0.2301,E1 3.7309,E2 464.2817} C_DIS
LIN {X 137.1927,Y -32.1669,Z 184,A -9.2251,B 3.569,C 0.2272,E1 3.7322,E2 462.3073} C_DIS
LIN {X 138.2616,Y -27.2068,Z 184,A -7.1781,B 3.5694,C 0.2216,E1 3.7334,E2 460.2609} C_DIS
LIN {X 138.9333,Y -23.5284,Z 184,A -5.7339,B 3.5696,C 0.2182,E1 3.7341,E2 458.8256} C_DIS
LIN {X 139.6226,Y -19.0259,Z 184,A -3.9162,B 3.5699,C 0.2135,E1 3.7348,E2 457.0112} C_DIS
LIN {X 140.0701,Y -15.3761,Z 184,A -2.5095,B 3.5701,C 0.2103,E1 3.7353,E2 455.6152} C_DIS
LIN {X 140.4229,Y -11.7214,Z 184,A -1.0993,B 3.5703,C 0.207,E1 3.7356,E2 454.215} C_DIS
LIN {X 140.7017,Y -7.7089,Z 184,A 0.5516,B 3.5705,C 0.2022,E1 3.7359,E2 452.5609} C_DIS
LIN {X 140.856,Y -3.9469,Z 184,A 2.0281,B 3.5707,C 0.1985,E1 3.736,E2 451.0906} C_DIS
LIN {X 140.9106,Y 0.4864,Z 184,A 3.6285,B 3.5709,C 0.1957,E1 3.736,E2 449.5158} C_DIS
LIN {X 140.8653,Y 3.6133,Z 184,A 4.9178,B 3.5711,C 0.1919,E1 3.736,E2 448.2233} C_DIS
LIN {X 140.7239,Y 7.266,Z 184,A 6.3487,B 3.5713,C 0.1884,E1 3.7358,E2 446.7987} C_DIS
LIN {X 140.4665,Y 11.2057,Z 184,A 7.9259,B 3.5715,C 0.1842,E1 3.7355,E2 445.2243} C_DIS
LIN {X 140.0832,Y 15.2543,Z 184,A 9.506,B 3.5717,C 0.1803,E1 3.735,E2 443.6529} C_DIS
LIN {X 139.5502,Y 19.5407,Z 184,A 11.1132,B 3.5719,C 0.1771,E1 3.7345,E2 442.0643} C_DIS
LIN {X 139.0803,Y 22.6474,Z 184,A 12.6586,B 3.5722,C 0.1705,E1 3.7338,E2 440.4828} C_DIS
LIN {X 138.5083,Y 25.9168,Z 184,A 14.0864,B 3.5724,C 0.1659,E1 3.733,E2 439.0439} C_DIS
LIN {X 137.7166,Y 29.8339,Z 184,A 15.7259,B 3.5726,C 0.1612,E1 3.732,E2 437.4014} C_DIS
LIN {X 136.6835,Y 34.2592,Z 184,A 16.8722,B 3.5725,C 0.1641,E1 3.7314,E2 436.3467} C_DIS
LIN {X 135.2809,Y 39.4335,Z 184,A 19.1971,B 3.5728,C 0.1565,E1 3.7296,E2 434.0016} C_DIS
LIN {X 133.9783,Y 43.6621,Z 184,A 20.9987,B 3.573,C 0.1516,E1 3.7281,E2 432.1989} C_DIS
LIN {X 132.7378,Y 47.295,Z 184,A 22.427,B 3.5731,C 0.1489,E1 3.7268,E2 430.7872} C_DIS
LIN {X 131.4701,Y 50.711,Z 184,A 23.7924,B 3.5733,C 0.1463,E1 3.7254,E2 429.4363} C_DIS
LIN {X 130.1641,Y 53.9749,Z 184,A 25.1662,B 3.5733,C 0.1432,E1 3.724,E2 428.069} C_DIS
LIN {X 128.7591,Y 57.2454,Z 184,A 26.5775,B 3.5735,C 0.1398,E1 3.7224,E2 426.6619} C_DIS
LIN {X 127.2729,Y 60.4775,Z 184,A 27.9907,B 3.5736,C 0.1364,E1 3.7207,E2 425.2523} C_DIS
LIN {X 125.69,Y 63.7017,Z 184,A 29.4263,B 3.5738,C 0.133,E1 3.7189,E2 423.8194} C_DIS
LIN {X 123.888,Y 67.144,Z 184,A 31.0225,B 3.5739,C 0.1289,E1 3.7168,E2 422.2205} C_DIS
LIN {X 121.6342,Y 71.1449,Z 184,A 32.8035,B 3.5741,C 0.1252,E1 3.7144,E2 420.4501} C_DIS
LIN {X 119.2863,Y 75.015,Z 184,A 34.5855,B 3.5741,C 0.1214,E1 3.7118,E2 418.6751} C_DIS
LIN {X 116.7794,Y 78.8606,Z 184,A 36.389,B 3.5743,C 0.1176,E1 3.709,E2 416.8792} C_DIS
LIN {X 114.0666,Y 82.7358,Z 184,A 38.2146,B 3.5744,C 0.1142,E1 3.706,E2 415.0657} C_DIS
LIN {X 111.9574,Y 85.5683,Z 184,A 39.9558,B 3.5746,C 0.1077,E1 3.703,E2 413.2845} C_DIS
LIN {X 109.378,Y 88.8427,Z 184,A 41.2997,B 3.5746,C 0.1076,E1 3.7008,E2 411.9858} C_DIS
LIN {X 106.3958,Y 92.3928,Z 184,A 43.049,B 3.5747,C 0.1049,E1 3.6976,E2 410.2536} C_DIS
LIN {X 103.6723,Y 95.4382,Z 184,A 44.687,B 3.5748,C 0.1016,E1 3.6945,E2 408.6183} C_DIS
LIN {X 100.6089,Y 98.6623,Z 184,A 46.4562,B 3.5748,C 0.0983,E1 3.6911,E2 406.8538} C_DIS
LIN {X 96.9977,Y 102.2156,Z 184,A 48.8261,B 3.5751,C 0.091,E1 3.6863,E2 404.4436} C_DIS
LIN {X 93.8831,Y 105.0828,Z 184,A 50.1289,B 3.5751,C 0.0919,E1 3.6837,E2 403.1945} C_DIS
LIN {X 90.4673,Y 108.0374,Z 184,A 51.9587,B 3.5751,C 0.0885,E1 3.6798,E2 401.3654} C_DIS
LIN {X 86.7322,Y 111.0589,Z 184,A 53.8533,B 3.5752,C 0.0856,E1 3.6756,E2 399.4782} C_DIS
LIN {X 83.1173,Y 113.7896,Z 184,A 55.9043,B 3.5753,C 0.0803,E1 3.671,E2 397.4004} C_DIS
LIN {X 80.0552,Y 115.9643,Z 184,A 57.1614,B 3.5753,C 0.0803,E1 3.6682,E2 396.1778} C_DIS
LIN {X 76.1838,Y 118.5432,Z 184,A 58.9794,B 3.5753,C 0.0781,E1 3.6639,E2 394.3692} C_DIS
LIN {X 72.3479,Y 120.9225,Z 184,A 60.7951,B 3.5755,C 0.0754,E1 3.6596,E2 392.5561} C_DIS
LIN {X 68.3244,Y 123.2404,Z 184,A 62.622,B 3.5755,C 0.0733,E1 3.6552,E2 390.737} C_DIS
LIN {X 65.368,Y 124.8314,Z 184,A 64.1773,B 3.5755,C 0.0696,E1 3.6513,E2 389.1575} C_DIS
LIN {X 62.299,Y 126.3909,Z 184,A 65.2589,B 3.5755,C 0.0707,E1 3.6487,E2 388.1166} C_DIS
LIN {X 59.333,Y 127.8103,Z 184,A 66.5583,B 3.5755,C 0.0693,E1 3.6454,E2 386.8221} C_DIS
LIN {X 55.998,Y 129.3061,Z 184,A 67.9491,B 3.5755,C 0.0684,E1 3.6419,E2 385.4437} C_DIS
LIN {X 53.2757,Y 130.4529,Z 184,A 69.2791,B 3.5756,C 0.0658,E1 3.6384,E2 384.0975} C_DIS
LIN {X 49.8609,Y 131.7952,Z 184,A 70.7114,B 3.5756,C 0.0647,E1 3.6347,E2 382.673} C_DIS
LIN {X 46.6545,Y 132.9643,Z 184,A 72.3417,B 3.5757,C 0.0611,E1 3.6303,E2 381.0121} C_DIS
LIN {X 43.4003,Y 134.0619,Z 184,A 73.8445,B 3.5757,C 0.0588,E1 3.6263,E2 379.4961} C_DIS
LIN {X 39.517,Y 135.2564,Z 184,A 75.0715,B 3.5757,C 0.0612,E1 3.6231,E2 378.3235} C_DIS
LIN {X 35.8456,Y 136.2763,Z 184,A 76.857,B 3.5757,C 0.0578,E1 3.6182,E2 376.5084} C_DIS
LIN {X 32.6927,Y 137.0664,Z 184,A 77.9133,B 3.5757,C 0.0591,E1 3.6155,E2 375.4861} C_DIS
LIN {X 28.788,Y 137.9408,Z 184,A 79.5538,B 3.5757,C 0.0579,E1 3.611,E2 373.8444} C_DIS
LIN {X 25.1275,Y 138.6529,Z 184,A 80.9688,B 3.5757,C 0.0579,E1 3.6071,E2 372.4425} C_DIS
LIN {X 19.9168,Y 139.4965,Z 184,A 83.1967,B 3.5758,C 0.056,E1 3.6009,E2 370.2051} C_DIS
LIN {X 15.3694,Y 140.0708,Z 184,A 85.0035,B 3.5758,C 0.0557,E1 3.5959,E2 368.4061} C_DIS
LIN {X 11.7752,Y 140.4184,Z 184,A 86.4448,B 3.5758,C 0.0554,E1 3.5919,E2 366.9688} C_DIS
LIN {X 7.7569,Y 140.6993,Z 184,A 88.2224,B 3.5758,C 0.0538,E1 3.5869,E2 365.1743} C_DIS
LIN {X 3.087,Y 140.8795,Z 184,A 90.1152,B 3.5758,C 0.0535,E1 3.5816,E2 363.2831} C_DIS
LIN {X -0.965,Y 140.9082,Z 184,A 91.6345,B 3.5758,C 0.0544,E1 3.5774,E2 361.7807} C_DIS
LIN {X -5.1015,Y 140.8195,Z 184,A 93.2693,B 3.5758,C 0.0547,E1 3.5729,E2 360.1527} C_DIS
LIN {X -12.1951,Y 140.3829,Z 184,A 96.2051,B 3.5758,C 0.0547,E1 3.5647,E2 357.2125} C_DIS
LIN {X -16.1448,Y 139.9843,Z 184,A 97.8657,B 3.5758,C 0.0547,E1 3.5601,E2 355.5468} C_DIS
LIN {X -19.8848,Y 139.501,Z 184,A 99.7885,B 3.5758,C 0.0521,E1 3.5546,E2 353.5756} C_DIS
LIN {X -24.0735,Y 138.8411,Z 184,A 101.2717,B 3.5758,C 0.0546,E1 3.5506,E2 352.1239} C_DIS
LIN {X -31.8342,Y 137.2687,Z 184,A 104.3432,B 3.5758,C 0.0573,E1 3.5423,E2 349.0729} C_DIS
LIN {X -35.247,Y 136.4328,Z 184,A 106.077,B 3.5758,C 0.0559,E1 3.5375,E2 347.3014} C_DIS
LIN {X -38.5495,Y 135.5368,Z 184,A 107.3143,B 3.5758,C 0.058,E1 3.5342,E2 346.0844} C_DIS
LIN {X -42.6759,Y 134.2933,Z 184,A 108.9723,B 3.5758,C 0.0599,E1 3.5298,E2 344.4394} C_DIS
LIN {X -45.8557,Y 133.2412,Z 184,A 110.5585,B 3.5758,C 0.0595,E1 3.5255,E2 342.8256} C_DIS
LIN {X -51.8797,Y 131.0156,Z 184,A 113.4327,B 3.5758,C 0.0601,E1 3.518,E2 339.9198} C_DIS
LIN {X -55.6676,Y 129.449,Z 184,A 114.6604,B 3.5757,C 0.0648,E1 3.515,E2 338.7489} C_DIS
LIN {X -58.3095,Y 128.2832,Z 184,A 116.7258,B 3.5757,C 0.0601,E1 3.5095,E2 336.571} C_DIS
LIN {X -64.0472,Y 125.5141,Z 184,A 118.4685,B 3.5756,C 0.0688,E1 3.5053,E2 334.938} C_DIS
LIN {X -67.2154,Y 123.849,Z 184,A 120.0967,B 3.5756,C 0.0695,E1 3.5013,E2 333.2889} C_DIS
LIN {X -70.2084,Y 122.1777,Z 184,A 122.1681,B 3.5756,C 0.067,E1 3.4961,E2 331.1322} C_DIS
LIN {X -75.2771,Y 119.1208,Z 184,A 123.8055,B 3.5755,C 0.0754,E1 3.4924,E2 329.5946} C_DIS
LIN {X -79.3733,Y 116.4323,Z 184,A 126.012,B 3.5755,C 0.077,E1 3.4872,E2 327.3625} C_DIS
LIN {X -82.0342,Y 114.5723,Z 184,A 127.5486,B 3.5755,C 0.0777,E1 3.4837,E2 325.7993} C_DIS
LIN {X -84.8058,Y 112.5362,Z 184,A 128.7574,B 3.5753,C 0.0812,E1 3.481,E2 324.6157} C_DIS
LIN {X -88.3918,Y 109.7419,Z 184,A 130.6203,B 3.5753,C 0.0842,E1 3.4769,E2 322.7524} C_DIS
LIN {X -91.6099,Y 107.0711,Z 184,A 132.4111,B 3.5752,C 0.0867,E1 3.4731,E2 320.9514} C_DIS
LIN {X -95.7446,Y 103.3901,Z 184,A 134.7498,B 3.5752,C 0.0903,E1 3.4682,E2 318.6033} C_DIS
LIN {X -99.0138,Y 100.2639,Z 184,A 136.5474,B 3.575,C 0.0941,E1 3.4646,E2 316.8123} C_DIS
LIN {X -101.8667,Y 97.3631,Z 184,A 138.3029,B 3.575,C 0.0968,E1 3.4612,E2 315.0452} C_DIS
LIN {X -106.808,Y 91.9155,Z 184,A 141.3626,B 3.5748,C 0.1026,E1 3.4555,E2 311.9791} C_DIS
LIN {X -108.6633,Y 89.7147,Z 184,A 142.6999,B 3.5748,C 0.1042,E1 3.4531,E2 310.6214} C_DIS
LIN {X -111.7676,Y 85.8165,Z 184,A 144.7151,B 3.5746,C 0.1087,E1 3.4496,E2 308.6092} C_DIS
LIN {X -114.554,Y 82.0598,Z 184,A 146.5774,B 3.5745,C 0.1132,E1 3.4466,E2 306.7534} C_DIS
LIN {X -118.6949,Y 75.9469,Z 184,A 149.742,B 3.5743,C 0.1193,E1 3.4417,E2 303.5705} C_DIS
LIN {X -121.1278,Y 72.0034,Z 184,A 151.6654,B 3.5741,C 0.1236,E1 3.4389,E2 301.6436} C_DIS
LIN {X -122.8397,Y 69.0421,Z 184,A 153.2194,B 3.5741,C 0.1261,E1 3.4367,E2 300.0697} C_DIS
LIN {X -125.2391,Y 64.5876,Z 184,A 155.3034,B 3.5738,C 0.1311,E1 3.434,E2 297.9839} C_DIS
LIN {X -127.0024,Y 61.0438,Z 184,A 156.8102,B 3.5737,C 0.1357,E1 3.4321,E2 296.4915} C_DIS
LIN {X -128.472,Y 57.8872,Z 184,A 158.3449,B 3.5736,C 0.1387,E1 3.4303,E2 294.9427} C_DIS
LIN {X -129.9255,Y 54.5462,Z 184,A 159.8421,B 3.5734,C 0.1425,E1 3.4287,E2 293.4446} C_DIS
LIN {X -131.183,Y 51.4494,Z 184,A 161.2352,B 3.5733,C 0.1458,E1 3.4273,E2 292.0482} C_DIS
LIN {X -132.4635,Y 48.0559,Z 184,A 162.7973,B 3.5731,C 0.1493,E1 3.4257,E2 290.4759} C_DIS
LIN {X -133.5838,Y 44.8481,Z 184,A 164.2512,B 3.573,C 0.1526,E1 3.4244,E2 289.0137} C_DIS
LIN {X -134.6646,Y 41.4896,Z 184,A 165.5943,B 3.5728,C 0.1569,E1 3.4233,E2 287.6836} C_DIS
LIN {X -135.6233,Y 38.24,Z 184,A 167.1842,B 3.5727,C 0.1596,E1 3.422,E2 286.0673} C_DIS
LIN {X -136.5715,Y 34.7004,Z 184,A 168.7079,B 3.5725,C 0.1635,E1 3.421,E2 284.5403} C_DIS
LIN {X -137.2464,Y 31.932,Z 184,A 170.0727,B 3.5725,C 0.1656,E1 3.4201,E2 283.1496} C_DIS
LIN {X -138.4721,Y 26.1062,Z 184,A 172.5417,B 3.5721,C 0.1721,E1 3.4187,E2 280.6761} C_DIS
LIN {X -139.8025,Y 17.6539,Z 184,A 176.2786,B 3.5717,C 0.1805,E1 3.4172,E2 276.9082} C_DIS
LIN {X -140.3018,Y 13.0958,Z 184,A 178.1436,B 3.5714,C 0.1858,E1 3.4166,E2 275.0445} C_DIS
LIN {X -140.6138,Y 9.1651,Z 184,A -179.8294,B 3.5714,C 0.1881,E1 3.4163,E2 272.9628} C_DIS
LIN {X -140.8312,Y 4.7938,Z 184,A -178.1139,B 3.571,C 0.1935,E1 3.4161,E2 271.2571} C_DIS
LIN {X -140.9067,Y 1.2393,Z 184,A -176.851,B 3.5707,C 0.1985,E1 3.4161,E2 270.0193} C_DIS
LIN {X -140.8804,Y -3.0344,Z 184,A -175.0765,B 3.5705,C 0.2032,E1 3.4161,E2 268.241} C_DIS
LIN {X -140.7918,Y -5.8101,Z 184,A -173.3866,B 3.5705,C 0.2036,E1 3.4164,E2 266.4778} C_DIS
LIN {X -140.5084,Y -10.6551,Z 184,A -172.0043,B 3.57,C 0.2121,E1 3.4166,E2 265.1749} C_DIS
LIN {X -139.7583,Y -17.9907,Z 184,A -168.9589,B 3.5695,C 0.2203,E1 3.4175,E2 262.1255} C_DIS
Enddeposition()
END
